Yaskawa INFORM job: A_ROOF_UPPER_0614_2_PAINT_67.JBI

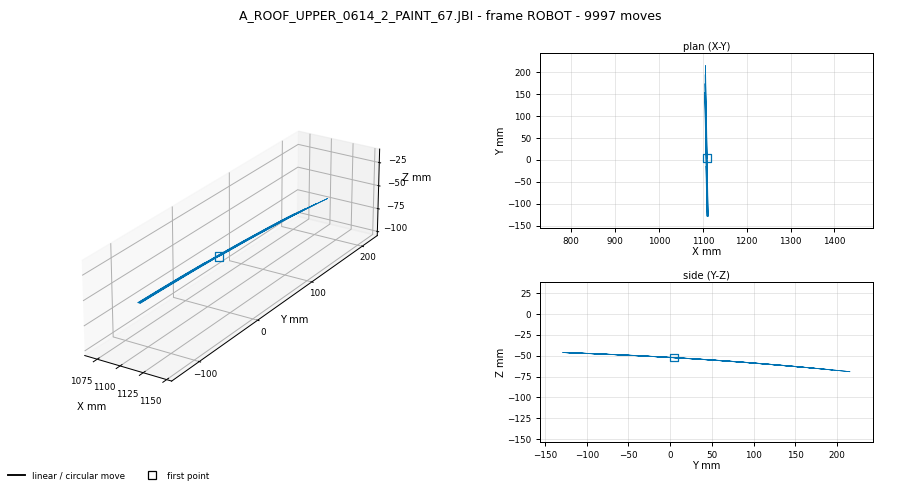
[picture p0: tool path of A_ROOF_UPPER_0614_2_PAINT_67.JBI in frame ROBOT, 9997 of 9997 moves have a stored position in this frame; points joined in program order, loops and branches not executed]
/JOB
//NAME A_ROOF_UPPER_0614_2_PAINT67
//POS
///NPOS 9997,0,0,0,0,0
///TOOL 1
///USER 0
///POSTYPE ROBOT
///RECTAN
///RCONF 1,0,0,0,0,0,0,0,0,0,0,0,0,0,0,0,0,0,0,0,0,0,0,0
C00000=1109.941,4.265,-52.087,179.831,6.526,149.242
C00001=1109.936,4.515,-52.102,179.832,6.531,149.243
C00002=1109.930,4.764,-52.116,179.832,6.536,149.244
C00003=1109.925,5.013,-52.130,179.833,6.541,149.244
C00004=1109.920,5.262,-52.145,179.834,6.545,149.245
C00005=1109.916,5.512,-52.159,179.834,6.550,149.246
C00006=1109.911,5.762,-52.173,179.835,6.554,149.247
C00007=1109.905,6.011,-52.189,179.835,6.559,149.248
C00008=1109.900,6.261,-52.203,179.836,6.564,149.249
C00009=1109.895,6.511,-52.218,179.837,6.568,149.249
C00010=1109.890,6.760,-52.232,179.837,6.573,149.250
C00011=1109.886,7.009,-52.247,179.837,6.577,149.251
C00012=1109.881,7.259,-52.261,179.838,6.581,149.252
C00013=1109.875,7.509,-52.276,179.838,6.586,149.253
C00014=1109.870,7.758,-52.291,179.840,6.590,149.254
C00015=1109.865,8.008,-52.305,179.840,6.595,149.254
C00016=1109.860,8.256,-52.320,179.841,6.600,149.255
C00017=1109.854,8.506,-52.335,179.841,6.605,149.256
C00018=1109.851,8.721,-52.347,179.842,6.609,149.257
C00019=1109.847,8.936,-52.360,179.842,6.613,149.258
C00020=1109.842,9.149,-52.373,179.843,6.616,149.258
C00021=1109.838,9.364,-52.385,179.843,6.620,149.259
C00022=1109.834,9.578,-52.397,179.843,6.625,149.260
C00023=1109.829,9.792,-52.411,179.844,6.628,149.261
C00024=1109.825,10.006,-52.423,179.844,6.632,149.261
C00025=1109.821,10.221,-52.436,179.845,6.636,149.262
C00026=1109.816,10.470,-52.451,179.845,6.640,149.263
C00027=1109.811,10.720,-52.465,179.846,6.645,149.264
C00028=1109.806,10.969,-52.480,179.846,6.649,149.265
C00029=1109.800,11.219,-52.495,179.847,6.654,149.266
C00030=1109.795,11.469,-52.510,179.847,6.659,149.266
C00031=1109.791,11.718,-52.525,179.847,6.663,149.267
C00032=1109.785,11.968,-52.539,179.848,6.667,149.268
C00033=1109.780,12.217,-52.554,179.849,6.672,149.269
C00034=1109.776,12.466,-52.569,179.850,6.676,149.270
C00035=1109.770,12.716,-52.584,179.850,6.681,149.271
C00036=1109.765,12.965,-52.599,179.850,6.685,149.272
C00037=1109.760,13.215,-52.614,179.851,6.689,149.272
C00038=1109.755,13.464,-52.629,179.852,6.694,149.273
C00039=1109.750,13.714,-52.643,179.852,6.699,149.274
C00040=1109.745,13.963,-52.658,179.853,6.703,149.275
C00041=1109.740,14.213,-52.673,179.853,6.707,149.275
C00042=1109.735,14.462,-52.688,179.854,6.712,149.276
C00043=1109.730,14.711,-52.703,179.854,6.716,149.277
C00044=1109.725,14.961,-52.718,179.855,6.721,149.278
C00045=1109.721,15.211,-52.733,179.856,6.725,149.279
C00046=1109.715,15.460,-52.749,179.856,6.729,149.280
C00047=1109.710,15.710,-52.763,179.856,6.734,149.281
C00048=1109.705,15.959,-52.779,179.857,6.738,149.281
C00049=1109.700,16.209,-52.794,179.858,6.743,149.282
C00050=1109.695,16.458,-52.808,179.859,6.747,149.283
C00051=1109.690,16.708,-52.824,179.859,6.751,149.284
C00052=1109.685,16.957,-52.839,179.860,6.756,149.285
C00053=1109.680,17.207,-52.854,179.861,6.760,149.285
C00054=1109.675,17.456,-52.869,179.861,6.765,149.286
C00055=1109.670,17.706,-52.885,179.862,6.770,149.287
C00056=1109.665,17.956,-52.899,179.862,6.773,149.288
C00057=1109.660,18.205,-52.914,179.863,6.778,149.288
C00058=1109.655,18.454,-52.929,179.864,6.782,149.289
C00059=1109.650,18.704,-52.945,179.864,6.787,149.290
C00060=1109.645,18.953,-52.959,179.865,6.790,149.291
C00061=1109.639,19.203,-52.975,179.865,6.795,149.292
C00062=1109.635,19.452,-52.990,179.866,6.799,149.292
C00063=1109.630,19.702,-53.006,179.867,6.804,149.293
C00064=1109.625,19.951,-53.021,179.867,6.809,149.294
C00065=1109.620,20.201,-53.036,179.868,6.812,149.295
C00066=1109.615,20.450,-53.051,179.868,6.817,149.296
C00067=1109.610,20.700,-53.066,179.869,6.821,149.296
C00068=1109.605,20.949,-53.081,179.871,6.826,149.297
C00069=1109.600,21.199,-53.097,179.870,6.830,149.298
C00070=1109.596,21.448,-53.112,179.872,6.834,149.298
C00071=1109.590,21.697,-53.128,179.872,6.839,149.299
C00072=1109.584,21.947,-53.143,179.873,6.843,149.300
C00073=1109.580,22.196,-53.158,179.874,6.848,149.301
C00074=1109.575,22.411,-53.171,179.874,6.851,149.301
C00075=1109.572,22.625,-53.184,179.875,6.855,149.302
C00076=1109.567,22.840,-53.197,179.875,6.858,149.303
C00077=1109.562,23.053,-53.211,179.876,6.863,149.303
C00078=1109.559,23.267,-53.224,179.877,6.866,149.304
C00079=1109.555,23.482,-53.238,179.877,6.869,149.305
C00080=1109.549,23.696,-53.250,179.878,6.873,149.305
C00081=1109.546,23.910,-53.263,179.878,6.876,149.306
C00082=1109.540,24.159,-53.279,179.879,6.881,149.307
C00083=1109.536,24.409,-53.295,179.880,6.885,149.307
C00084=1109.531,24.658,-53.310,179.881,6.890,149.308
C00085=1109.526,24.908,-53.326,179.882,6.894,149.309
C00086=1109.520,25.157,-53.341,179.882,6.898,149.310
C00087=1109.516,25.407,-53.356,179.883,6.902,149.310
C00088=1109.511,25.656,-53.372,179.884,6.907,149.311
C00089=1109.505,25.906,-53.388,179.885,6.911,149.312
C00090=1109.501,26.155,-53.403,179.885,6.915,149.312
C00091=1109.496,26.405,-53.419,179.886,6.919,149.313
C00092=1109.491,26.654,-53.434,179.887,6.924,149.314
C00093=1109.486,26.903,-53.449,179.888,6.928,149.315
C00094=1109.481,27.153,-53.465,179.888,6.932,149.315
C00095=1109.476,27.402,-53.481,179.889,6.936,149.316
C00096=1109.471,27.652,-53.497,179.890,6.941,149.317
C00097=1109.466,27.901,-53.512,179.891,6.945,149.317
C00098=1109.461,28.151,-53.528,179.892,6.949,149.318
C00099=1109.456,28.400,-53.544,179.892,6.953,149.319
C00100=1109.450,28.650,-53.559,179.893,6.957,149.320
C00101=1109.446,28.900,-53.574,179.894,6.962,149.320
C00102=1109.441,29.149,-53.590,179.895,6.966,149.321
C00103=1109.436,29.398,-53.606,179.895,6.970,149.322
C00104=1109.431,29.647,-53.622,179.896,6.974,149.323
C00105=1109.427,29.897,-53.637,179.897,6.979,149.323
C00106=1109.421,30.146,-53.653,179.898,6.983,149.324
C00107=1109.416,30.396,-53.669,179.899,6.986,149.324
C00108=1109.411,30.645,-53.685,179.899,6.991,149.325
C00109=1109.406,30.895,-53.701,179.900,6.995,149.326
C00110=1109.402,31.144,-53.716,179.901,7.000,149.327
C00111=1109.396,31.394,-53.732,179.902,7.003,149.327
C00112=1109.391,31.643,-53.747,179.903,7.007,149.328
C00113=1109.387,31.893,-53.764,179.904,7.012,149.329
C00114=1109.381,32.142,-53.780,179.905,7.016,149.329
C00115=1109.376,32.392,-53.795,179.905,7.020,149.330
C00116=1109.371,32.641,-53.812,179.906,7.024,149.331
C00117=1109.367,32.890,-53.827,179.907,7.029,149.331
C00118=1109.362,33.140,-53.843,179.908,7.033,149.332
C00119=1109.356,33.390,-53.858,179.909,7.037,149.333
C00120=1109.351,33.638,-53.875,179.910,7.041,149.333
C00121=1109.347,33.888,-53.891,179.911,7.045,149.334
C00122=1109.341,34.138,-53.906,179.912,7.049,149.335
C00123=1109.337,34.387,-53.923,179.913,7.054,149.335
C00124=1109.331,34.637,-53.938,179.913,7.057,149.336
C00125=1109.326,34.886,-53.955,179.914,7.061,149.337
C00126=1109.322,35.136,-53.971,179.915,7.066,149.337
C00127=1109.317,35.385,-53.986,179.916,7.070,149.338
C00128=1109.312,35.634,-54.002,179.917,7.074,149.339
C00129=1109.307,35.884,-54.018,179.918,7.078,149.339
C00130=1109.303,36.098,-54.032,179.918,7.081,149.340
C00131=1109.299,36.312,-54.046,179.919,7.086,149.341
C00132=1109.294,36.526,-54.060,179.920,7.089,149.341
C00133=1109.290,36.740,-54.073,179.921,7.092,149.342
C00134=1109.285,36.954,-54.087,179.922,7.096,149.342
C00135=1109.281,37.168,-54.101,179.923,7.100,149.343
C00136=1109.277,37.382,-54.115,179.924,7.103,149.343
C00137=1109.273,37.596,-54.129,179.924,7.106,149.344
C00138=1109.267,37.846,-54.144,179.925,7.111,149.345
C00139=1109.263,38.095,-54.161,179.926,7.115,149.345
C00140=1109.257,38.345,-54.177,179.927,7.119,149.346
C00141=1109.253,38.594,-54.193,179.928,7.123,149.347
C00142=1109.248,38.843,-54.209,179.929,7.127,149.347
C00143=1109.243,39.093,-54.225,179.930,7.132,149.348
C00144=1109.238,39.342,-54.241,179.930,7.135,149.349
C00145=1109.233,39.592,-54.258,179.932,7.139,149.349
C00146=1109.228,39.841,-54.274,179.933,7.143,149.350
C00147=1109.223,40.091,-54.290,179.934,7.148,149.350
C00148=1109.218,40.339,-54.306,179.935,7.151,149.351
C00149=1109.213,40.590,-54.322,179.936,7.155,149.352
C00150=1109.208,40.839,-54.339,179.937,7.160,149.352
C00151=1109.203,41.088,-54.356,179.938,7.164,149.353
C00152=1109.198,41.338,-54.372,179.938,7.168,149.354
C00153=1109.193,41.587,-54.388,179.939,7.172,149.354
C00154=1109.188,41.837,-54.404,179.940,7.176,149.355
C00155=1109.183,42.086,-54.420,179.942,7.180,149.355
C00156=1109.179,42.335,-54.437,179.943,7.184,149.356
C00157=1109.174,42.585,-54.453,179.944,7.188,149.357
C00158=1109.169,42.834,-54.469,179.945,7.192,149.357
C00159=1109.163,43.083,-54.486,179.946,7.196,149.358
C00160=1109.159,43.333,-54.503,179.947,7.201,149.359
C00161=1109.154,43.583,-54.519,179.948,7.204,149.359
C00162=1109.149,43.832,-54.535,179.949,7.208,149.360
C00163=1109.144,44.081,-54.552,179.950,7.213,149.360
C00164=1109.139,44.331,-54.567,179.951,7.217,149.361
C00165=1109.134,44.580,-54.585,179.951,7.220,149.362
C00166=1109.129,44.830,-54.601,179.953,7.224,149.362
C00167=1109.124,45.079,-54.618,179.954,7.229,149.363
C00168=1109.120,45.328,-54.634,179.955,7.233,149.363
C00169=1109.114,45.578,-54.650,179.956,7.237,149.364
C00170=1109.109,45.827,-54.667,179.957,7.241,149.365
C00171=1109.105,46.077,-54.684,179.958,7.245,149.365
C00172=1109.100,46.326,-54.700,179.959,7.249,149.366
C00173=1109.095,46.575,-54.717,179.960,7.253,149.366
C00174=1109.089,46.825,-54.733,179.961,7.257,149.367
C00175=1109.085,47.074,-54.750,179.962,7.261,149.367
C00176=1109.080,47.324,-54.766,179.963,7.265,149.368
C00177=1109.075,47.573,-54.783,179.964,7.269,149.369
C00178=1109.070,47.822,-54.800,179.966,7.273,149.369
C00179=1109.065,48.072,-54.816,179.966,7.277,149.370
C00180=1109.060,48.321,-54.833,179.968,7.281,149.371
C00181=1109.056,48.570,-54.849,179.969,7.285,149.371
C00182=1109.050,48.820,-54.867,179.970,7.289,149.372
C00183=1109.045,49.069,-54.883,179.971,7.293,149.372
C00184=1109.041,49.318,-54.900,179.972,7.297,149.373
C00185=1109.035,49.569,-54.916,179.973,7.301,149.373
C00186=1109.031,49.782,-54.931,179.974,7.304,149.374
C00187=1109.027,49.996,-54.945,179.975,7.308,149.374
C00188=1109.023,50.210,-54.959,179.976,7.311,149.375
C00189=1109.018,50.424,-54.974,179.977,7.315,149.376
C00190=1109.014,50.638,-54.988,179.978,7.318,149.376
C00191=1109.010,50.852,-55.003,179.979,7.322,149.376
C00192=1109.006,51.066,-55.016,179.980,7.325,149.377
C00193=1109.001,51.280,-55.031,179.981,7.329,149.377
C00194=1108.997,51.530,-55.048,179.982,7.333,149.378
C00195=1108.992,51.779,-55.065,179.983,7.337,149.379
C00196=1108.987,52.028,-55.082,179.984,7.340,149.379
C00197=1108.982,52.278,-55.098,179.985,7.344,149.380
C00198=1108.977,52.527,-55.116,179.986,7.349,149.380
C00199=1108.973,52.776,-55.133,179.988,7.352,149.381
C00200=1108.968,53.025,-55.149,179.989,7.357,149.381
C00201=1108.962,53.275,-55.166,179.989,7.360,149.382
C00202=1108.958,53.524,-55.183,179.991,7.364,149.382
C00203=1108.953,53.774,-55.200,179.992,7.368,149.383
C00204=1108.948,54.023,-55.217,179.994,7.372,149.384
C00205=1108.942,54.273,-55.234,179.995,7.377,149.384
C00206=1108.938,54.522,-55.251,179.995,7.380,149.385
C00207=1108.933,54.771,-55.269,179.997,7.384,149.385
C00208=1108.929,55.021,-55.285,179.998,7.388,149.386
C00209=1108.923,55.270,-55.302,179.999,7.392,149.386
C00210=1108.918,55.520,-55.319,-179.999,7.397,149.387
C00211=1108.913,55.769,-55.336,-179.999,7.400,149.387
C00212=1108.909,56.018,-55.354,-179.997,7.404,149.388
C00213=1108.904,56.268,-55.371,-179.996,7.408,149.389
C00214=1108.899,56.517,-55.387,-179.995,7.412,149.389
C00215=1108.893,56.767,-55.404,-179.994,7.416,149.390
C00216=1108.889,57.015,-55.422,-179.993,7.420,149.390
C00217=1108.884,57.265,-55.439,-179.992,7.424,149.391
C00218=1108.880,57.515,-55.456,-179.990,7.428,149.391
C00219=1108.874,57.764,-55.473,-179.989,7.432,149.392
C00220=1108.870,58.013,-55.490,-179.987,7.436,149.392
C00221=1108.864,58.262,-55.507,-179.986,7.440,149.393
C00222=1108.859,58.512,-55.524,-179.985,7.443,149.394
C00223=1108.855,58.761,-55.542,-179.984,7.448,149.394
C00224=1108.850,59.011,-55.559,-179.983,7.452,149.395
C00225=1108.845,59.260,-55.576,-179.982,7.456,149.395
C00226=1108.840,59.509,-55.593,-179.980,7.460,149.396
C00227=1108.834,59.759,-55.611,-179.980,7.463,149.396
C00228=1108.830,60.008,-55.627,-179.978,7.467,149.397
C00229=1108.825,60.257,-55.645,-179.977,7.472,149.397
C00230=1108.821,60.507,-55.662,-179.975,7.475,149.398
C00231=1108.816,60.756,-55.680,-179.974,7.480,149.399
C00232=1108.810,61.006,-55.697,-179.973,7.484,149.399
C00233=1108.806,61.255,-55.714,-179.972,7.487,149.400
C00234=1108.801,61.504,-55.732,-179.971,7.491,149.400
C00235=1108.796,61.754,-55.749,-179.970,7.495,149.401
C00236=1108.791,62.002,-55.766,-179.968,7.499,149.401
C00237=1108.786,62.252,-55.783,-179.966,7.503,149.402
C00238=1108.781,62.501,-55.801,-179.965,7.507,149.402
C00239=1108.776,62.751,-55.818,-179.964,7.511,149.403
C00240=1108.772,63.000,-55.836,-179.963,7.515,149.403
C00241=1108.766,63.250,-55.853,-179.962,7.519,149.404
C00242=1108.763,63.463,-55.868,-179.961,7.522,149.404
C00243=1108.759,63.678,-55.884,-179.959,7.526,149.405
C00244=1108.755,63.891,-55.898,-179.958,7.529,149.405
C00245=1108.750,64.105,-55.913,-179.957,7.532,149.405
C00246=1108.745,64.319,-55.928,-179.956,7.536,149.406
C00247=1108.742,64.533,-55.944,-179.955,7.539,149.407
C00248=1108.737,64.747,-55.959,-179.954,7.543,149.407
C00249=1108.733,64.961,-55.973,-179.953,7.546,149.407
C00250=1108.728,65.210,-55.991,-179.952,7.550,149.408
C00251=1108.723,65.460,-56.009,-179.951,7.554,149.409
C00252=1108.718,65.709,-56.026,-179.949,7.558,149.409
C00253=1108.714,65.958,-56.044,-179.948,7.562,149.409
C00254=1108.709,66.208,-56.061,-179.946,7.566,149.410
C00255=1108.704,66.457,-56.079,-179.945,7.570,149.410
C00256=1108.699,66.706,-56.097,-179.944,7.573,149.411
C00257=1108.695,66.955,-56.114,-179.943,7.577,149.412
C00258=1108.690,67.205,-56.132,-179.941,7.581,149.412
C00259=1108.685,67.454,-56.150,-179.940,7.585,149.413
C00260=1108.680,67.704,-56.167,-179.939,7.589,149.413
C00261=1108.675,67.953,-56.185,-179.937,7.593,149.414
C00262=1108.670,68.202,-56.203,-179.936,7.598,149.414
C00263=1108.665,68.451,-56.221,-179.935,7.601,149.415
C00264=1108.660,68.701,-56.238,-179.933,7.605,149.415
C00265=1108.655,68.950,-56.256,-179.932,7.609,149.416
C00266=1108.650,69.199,-56.274,-179.931,7.613,149.416
C00267=1108.646,69.448,-56.292,-179.929,7.617,149.417
C00268=1108.641,69.699,-56.309,-179.928,7.621,149.417
C00269=1108.636,69.948,-56.327,-179.926,7.625,149.418
C00270=1108.631,70.197,-56.345,-179.925,7.629,149.418
C00271=1108.626,70.446,-56.363,-179.924,7.632,149.419
C00272=1108.621,70.695,-56.381,-179.923,7.636,149.419
C00273=1108.616,70.945,-56.399,-179.921,7.640,149.420
C00274=1108.611,71.194,-56.416,-179.920,7.644,149.420
C00275=1108.607,71.443,-56.434,-179.919,7.648,149.421
C00276=1108.602,71.692,-56.452,-179.917,7.652,149.421
C00277=1108.597,71.942,-56.470,-179.916,7.656,149.422
C00278=1108.592,72.191,-56.488,-179.914,7.660,149.422
C00279=1108.588,72.441,-56.506,-179.913,7.664,149.423
C00280=1108.583,72.690,-56.524,-179.912,7.668,149.423
C00281=1108.578,72.939,-56.542,-179.911,7.672,149.424
C00282=1108.573,73.188,-56.560,-179.909,7.676,149.424
C00283=1108.568,73.437,-56.578,-179.908,7.680,149.425
C00284=1108.563,73.686,-56.596,-179.906,7.684,149.425
C00285=1108.558,73.936,-56.614,-179.905,7.688,149.426
C00286=1108.554,74.186,-56.632,-179.904,7.692,149.426
C00287=1108.549,74.435,-56.649,-179.902,7.696,149.427
C00288=1108.544,74.684,-56.667,-179.901,7.700,149.427
C00289=1108.539,74.933,-56.687,-179.899,7.704,149.428
C00290=1108.534,75.183,-56.705,-179.898,7.707,149.428
C00291=1108.529,75.432,-56.723,-179.897,7.711,149.429
C00292=1108.525,75.682,-56.741,-179.895,7.715,149.429
C00293=1108.520,75.931,-56.759,-179.894,7.719,149.430
C00294=1108.515,76.180,-56.777,-179.893,7.723,149.430
C00295=1108.510,76.429,-56.795,-179.891,7.727,149.431
C00296=1108.505,76.678,-56.813,-179.889,7.731,149.431
C00297=1108.501,76.928,-56.831,-179.888,7.735,149.432
C00298=1108.496,77.142,-56.847,-179.887,7.738,149.432
C00299=1108.492,77.355,-56.863,-179.886,7.741,149.433
C00300=1108.488,77.570,-56.878,-179.885,7.745,149.433
C00301=1108.483,77.783,-56.894,-179.885,7.748,149.434
C00302=1108.479,77.997,-56.910,-179.884,7.751,149.434
C00303=1108.475,78.211,-56.926,-179.883,7.754,149.435
C00304=1108.472,78.425,-56.941,-179.882,7.757,149.435
C00305=1108.467,78.638,-56.956,-179.881,7.760,149.435
C00306=1108.462,78.888,-56.974,-179.881,7.764,149.436
C00307=1108.457,79.138,-56.993,-179.879,7.768,149.437
C00308=1108.453,79.386,-57.012,-179.879,7.771,149.437
C00309=1108.448,79.635,-57.030,-179.877,7.775,149.438
C00310=1108.443,79.885,-57.048,-179.876,7.779,149.438
C00311=1108.438,80.134,-57.066,-179.875,7.783,149.439
C00312=1108.433,80.384,-57.085,-179.874,7.786,149.439
C00313=1108.428,80.633,-57.103,-179.873,7.790,149.440
C00314=1108.423,80.882,-57.121,-179.872,7.794,149.440
C00315=1108.419,81.132,-57.140,-179.871,7.798,149.441
C00316=1108.414,81.380,-57.158,-179.870,7.801,149.442
C00317=1108.409,81.630,-57.177,-179.869,7.805,149.442
C00318=1108.404,81.879,-57.195,-179.868,7.808,149.443
C00319=1108.400,82.129,-57.213,-179.867,7.813,149.443
C00320=1108.395,82.377,-57.232,-179.865,7.816,149.444
C00321=1108.389,82.627,-57.251,-179.865,7.820,149.444
C00322=1108.385,82.877,-57.269,-179.863,7.824,149.445
C00323=1108.380,83.125,-57.288,-179.863,7.827,149.445
C00324=1108.375,83.375,-57.306,-179.861,7.831,149.446
C00325=1108.370,83.625,-57.325,-179.861,7.835,149.446
C00326=1108.366,83.873,-57.343,-179.859,7.839,149.447
C00327=1108.361,84.122,-57.361,-179.858,7.843,149.448
C00328=1108.356,84.372,-57.381,-179.857,7.846,149.448
C00329=1108.351,84.621,-57.399,-179.856,7.850,149.449
C00330=1108.346,84.870,-57.417,-179.855,7.853,149.449
C00331=1108.342,85.120,-57.437,-179.853,7.857,149.450
C00332=1108.337,85.369,-57.455,-179.852,7.862,149.450
C00333=1108.332,85.617,-57.473,-179.851,7.865,149.451
C00334=1108.327,85.868,-57.492,-179.850,7.869,149.451
C00335=1108.322,86.116,-57.511,-179.848,7.873,149.452
C00336=1108.317,86.365,-57.529,-179.848,7.876,149.452
C00337=1108.312,86.616,-57.548,-179.846,7.880,149.453
C00338=1108.308,86.864,-57.566,-179.845,7.884,149.453
C00339=1108.303,87.114,-57.585,-179.844,7.888,149.454
C00340=1108.298,87.363,-57.604,-179.843,7.892,149.454
C00341=1108.293,87.612,-57.622,-179.841,7.895,149.455
C00342=1108.289,87.862,-57.642,-179.841,7.899,149.455
C00343=1108.284,88.110,-57.660,-179.839,7.903,149.456
C00344=1108.278,88.360,-57.679,-179.838,7.907,149.456
C00345=1108.274,88.609,-57.698,-179.837,7.910,149.457
C00346=1108.269,88.858,-57.716,-179.835,7.914,149.457
C00347=1108.265,89.108,-57.736,-179.834,7.918,149.458
C00348=1108.260,89.357,-57.754,-179.833,7.921,149.458
C00349=1108.255,89.606,-57.773,-179.832,7.925,149.459
C00350=1108.250,89.855,-57.792,-179.830,7.929,149.459
C00351=1108.245,90.104,-57.811,-179.829,7.933,149.460
C00352=1108.241,90.354,-57.830,-179.828,7.937,149.460
C00353=1108.235,90.603,-57.848,-179.826,7.941,149.461
C00354=1108.232,90.817,-57.865,-179.825,7.944,149.461
C00355=1108.228,91.031,-57.881,-179.824,7.947,149.462
C00356=1108.223,91.244,-57.897,-179.823,7.951,149.462
C00357=1108.219,91.458,-57.913,-179.822,7.954,149.463
C00358=1108.215,91.671,-57.929,-179.821,7.957,149.463
C00359=1108.211,91.885,-57.946,-179.820,7.960,149.463
C00360=1108.207,92.100,-57.962,-179.819,7.963,149.464
C00361=1108.203,92.313,-57.978,-179.817,7.967,149.464
C00362=1108.198,92.562,-57.998,-179.816,7.970,149.465
C00363=1108.193,92.811,-58.016,-179.815,7.974,149.465
C00364=1108.188,93.061,-58.036,-179.813,7.978,149.466
C00365=1108.184,93.310,-58.054,-179.812,7.982,149.466
C00366=1108.179,93.559,-58.074,-179.811,7.985,149.467
C00367=1108.174,93.808,-58.092,-179.809,7.989,149.467
C00368=1108.169,94.057,-58.112,-179.808,7.993,149.468
C00369=1108.164,94.307,-58.131,-179.806,7.997,149.468
C00370=1108.160,94.556,-58.150,-179.805,8.001,149.468
C00371=1108.154,94.805,-58.169,-179.804,8.004,149.469
C00372=1108.150,95.054,-58.188,-179.802,8.008,149.469
C00373=1108.145,95.303,-58.207,-179.801,8.012,149.470
C00374=1108.140,95.553,-58.227,-179.799,8.016,149.470
C00375=1108.135,95.802,-58.245,-179.798,8.020,149.471
C00376=1108.131,96.052,-58.265,-179.797,8.023,149.471
C00377=1108.125,96.300,-58.284,-179.795,8.027,149.472
C00378=1108.121,96.550,-58.303,-179.794,8.031,149.472
C00379=1108.117,96.799,-58.323,-179.792,8.035,149.473
C00380=1108.112,97.048,-58.341,-179.790,8.039,149.473
C00381=1108.107,97.297,-58.361,-179.789,8.042,149.473
C00382=1108.102,97.546,-58.380,-179.788,8.046,149.474
C00383=1108.097,97.796,-58.400,-179.786,8.049,149.474
C00384=1108.093,98.044,-58.419,-179.785,8.053,149.475
C00385=1108.088,98.294,-58.438,-179.783,8.057,149.475
C00386=1108.083,98.543,-58.458,-179.781,8.061,149.476
C00387=1108.078,98.792,-58.477,-179.780,8.064,149.476
C00388=1108.074,99.042,-58.496,-179.779,8.068,149.476
C00389=1108.068,99.290,-58.516,-179.777,8.072,149.477
C00390=1108.064,99.540,-58.535,-179.776,8.076,149.477
C00391=1108.060,99.789,-58.554,-179.774,8.080,149.478
C00392=1108.054,100.038,-58.574,-179.772,8.084,149.478
C00393=1108.050,100.288,-58.593,-179.770,8.087,149.478
C00394=1108.044,100.537,-58.612,-179.769,8.090,149.479
C00395=1108.040,100.786,-58.632,-179.768,8.094,149.479
C00396=1108.035,101.035,-58.651,-179.766,8.098,149.480
C00397=1108.030,101.284,-58.670,-179.765,8.102,149.480
C00398=1108.025,101.534,-58.690,-179.763,8.106,149.481
C00399=1108.021,101.783,-58.710,-179.761,8.109,149.481
C00400=1108.016,102.032,-58.728,-179.759,8.113,149.481
C00401=1108.012,102.281,-58.749,-179.758,8.117,149.482
C00402=1108.007,102.530,-58.769,-179.756,8.121,149.482
C00403=1108.002,102.779,-58.788,-179.755,8.124,149.483
C00404=1107.997,103.029,-58.807,-179.753,8.128,149.483
C00405=1107.992,103.279,-58.827,-179.751,8.131,149.483
C00406=1107.987,103.527,-58.846,-179.750,8.135,149.484
C00407=1107.983,103.776,-58.866,-179.748,8.139,149.484
C00408=1107.978,104.026,-58.886,-179.746,8.143,149.484
C00409=1107.973,104.275,-58.906,-179.745,8.147,149.485
C00410=1107.969,104.488,-58.923,-179.743,8.149,149.485
C00411=1107.965,104.702,-58.939,-179.742,8.153,149.485
C00412=1107.961,104.916,-58.956,-179.740,8.156,149.486
C00413=1107.957,105.130,-58.973,-179.739,8.159,149.486
C00414=1107.953,105.343,-58.990,-179.737,8.162,149.486
C00415=1107.949,105.556,-59.007,-179.736,8.165,149.487
C00416=1107.944,105.770,-59.024,-179.735,8.168,149.487
C00417=1107.941,105.984,-59.040,-179.733,8.172,149.487
C00418=1107.936,106.233,-59.061,-179.731,8.175,149.487
C00419=1107.931,106.482,-59.080,-179.729,8.179,149.488
C00420=1107.926,106.731,-59.100,-179.727,8.183,149.488
C00421=1107.922,106.980,-59.120,-179.726,8.186,149.489
C00422=1107.917,107.230,-59.140,-179.724,8.190,149.489
C00423=1107.912,107.479,-59.160,-179.722,8.193,149.489
C00424=1107.907,107.728,-59.179,-179.720,8.197,149.489
C00425=1107.902,107.977,-59.199,-179.719,8.201,149.490
C00426=1107.898,108.226,-59.219,-179.716,8.204,149.490
C00427=1107.893,108.476,-59.239,-179.715,8.208,149.490
C00428=1107.888,108.724,-59.259,-179.713,8.211,149.491
C00429=1107.883,108.974,-59.279,-179.711,8.215,149.491
C00430=1107.879,109.223,-59.299,-179.709,8.219,149.491
C00431=1107.874,109.472,-59.319,-179.707,8.222,149.492
C00432=1107.870,109.721,-59.339,-179.705,8.226,149.492
C00433=1107.865,109.971,-59.359,-179.703,8.230,149.492
C00434=1107.860,110.219,-59.379,-179.701,8.233,149.493
C00435=1107.855,110.468,-59.398,-179.700,8.237,149.493
C00436=1107.851,110.717,-59.419,-179.698,8.241,149.493
C00437=1107.845,110.967,-59.439,-179.696,8.244,149.493
C00438=1107.841,111.216,-59.459,-179.694,8.248,149.494
C00439=1107.836,111.466,-59.479,-179.693,8.251,149.494
C00440=1107.831,111.714,-59.499,-179.691,8.254,149.494
C00441=1107.826,111.964,-59.519,-179.689,8.258,149.495
C00442=1107.822,112.213,-59.539,-179.687,8.261,149.495
C00443=1107.818,112.462,-59.559,-179.685,8.264,149.495
C00444=1107.812,112.711,-59.580,-179.684,8.268,149.496
C00445=1107.808,112.960,-59.600,-179.682,8.272,149.496
C00446=1107.803,113.209,-59.620,-179.680,8.274,149.496
C00447=1107.798,113.459,-59.640,-179.679,8.278,149.497
C00448=1107.793,113.707,-59.660,-179.677,8.282,149.497
C00449=1107.789,113.956,-59.680,-179.676,8.285,149.497
C00450=1107.783,114.206,-59.701,-179.674,8.288,149.497
C00451=1107.779,114.455,-59.721,-179.672,8.292,149.498
C00452=1107.775,114.704,-59.741,-179.670,8.296,149.498
C00453=1107.770,114.953,-59.761,-179.668,8.299,149.498
C00454=1107.765,115.202,-59.781,-179.666,8.302,149.499
C00455=1107.760,115.452,-59.802,-179.665,8.306,149.499
C00456=1107.756,115.701,-59.823,-179.663,8.309,149.499
C00457=1107.751,115.950,-59.842,-179.661,8.312,149.499
C00458=1107.747,116.199,-59.863,-179.660,8.316,149.500
C00459=1107.741,116.448,-59.884,-179.658,8.319,149.500
C00460=1107.737,116.697,-59.904,-179.656,8.322,149.500
C00461=1107.732,116.946,-59.924,-179.654,8.326,149.501
C00462=1107.727,117.195,-59.944,-179.653,8.330,149.501
C00463=1107.722,117.444,-59.965,-179.651,8.332,149.501
C00464=1107.718,117.693,-59.985,-179.649,8.336,149.501
C00465=1107.713,117.942,-60.006,-179.647,8.340,149.502
C00466=1107.709,118.156,-60.023,-179.646,8.342,149.502
C00467=1107.705,118.370,-60.040,-179.645,8.345,149.502
C00468=1107.701,118.583,-60.058,-179.643,8.348,149.503
C00469=1107.697,118.797,-60.076,-179.642,8.351,149.503
C00470=1107.693,119.010,-60.094,-179.640,8.353,149.503
C00471=1107.688,119.224,-60.111,-179.638,8.357,149.503
C00472=1107.685,119.437,-60.128,-179.637,8.360,149.503
C00473=1107.681,119.650,-60.146,-179.635,8.362,149.504
C00474=1107.676,119.900,-60.167,-179.634,8.366,149.504
C00475=1107.671,120.149,-60.187,-179.632,8.369,149.504
C00476=1107.667,120.398,-60.207,-179.630,8.372,149.505
C00477=1107.661,120.647,-60.228,-179.629,8.376,149.505
C00478=1107.657,120.896,-60.249,-179.627,8.379,149.505
C00479=1107.652,121.146,-60.270,-179.625,8.382,149.505
C00480=1107.648,121.395,-60.290,-179.623,8.386,149.506
C00481=1107.643,121.644,-60.311,-179.622,8.389,149.506
C00482=1107.638,121.893,-60.332,-179.620,8.392,149.506
C00483=1107.634,122.142,-60.353,-179.618,8.396,149.507
C00484=1107.629,122.391,-60.374,-179.616,8.399,149.507
C00485=1107.625,122.640,-60.394,-179.615,8.403,149.507
C00486=1107.619,122.889,-60.415,-179.613,8.406,149.507
C00487=1107.615,123.138,-60.435,-179.611,8.409,149.508
C00488=1107.610,123.387,-60.456,-179.609,8.412,149.508
C00489=1107.605,123.636,-60.477,-179.608,8.416,149.508
C00490=1107.601,123.885,-60.497,-179.606,8.420,149.509
C00491=1107.596,124.135,-60.518,-179.604,8.422,149.509
C00492=1107.592,124.384,-60.539,-179.602,8.426,149.509
C00493=1107.587,124.633,-60.561,-179.600,8.430,149.509
C00494=1107.583,124.882,-60.581,-179.599,8.432,149.510
C00495=1107.577,125.131,-60.602,-179.597,8.436,149.510
C00496=1107.573,125.380,-60.622,-179.595,8.439,149.510
C00497=1107.568,125.629,-60.643,-179.594,8.443,149.511
C00498=1107.563,125.878,-60.664,-179.592,8.446,149.511
C00499=1107.558,126.127,-60.685,-179.590,8.450,149.511
C00500=1107.555,126.377,-60.706,-179.588,8.452,149.511
C00501=1107.549,126.626,-60.727,-179.586,8.456,149.512
C00502=1107.544,126.875,-60.748,-179.585,8.460,149.512
C00503=1107.540,127.123,-60.769,-179.583,8.462,149.512
C00504=1107.535,127.373,-60.790,-179.581,8.466,149.512
C00505=1107.531,127.622,-60.810,-179.579,8.469,149.513
C00506=1107.526,127.871,-60.832,-179.578,8.472,149.513
C00507=1107.521,128.120,-60.853,-179.576,8.476,149.513
C00508=1107.517,128.369,-60.874,-179.574,8.479,149.514
C00509=1107.511,128.618,-60.895,-179.572,8.482,149.514
C00510=1107.507,128.867,-60.916,-179.571,8.486,149.514
C00511=1107.502,129.116,-60.937,-179.569,8.490,149.514
C00512=1107.498,129.366,-60.958,-179.567,8.492,149.515
C00513=1107.493,129.614,-60.979,-179.565,8.496,149.515
C00514=1107.488,129.864,-61.000,-179.564,8.500,149.515
C00515=1107.483,130.112,-61.022,-179.562,8.503,149.516
C00516=1107.479,130.361,-61.042,-179.560,8.506,149.516
C00517=1107.474,130.611,-61.064,-179.558,8.509,149.516
C00518=1107.470,130.860,-61.085,-179.556,8.513,149.516
C00519=1107.464,131.109,-61.106,-179.555,8.516,149.517
C00520=1107.460,131.357,-61.127,-179.553,8.519,149.517
C00521=1107.456,131.607,-61.149,-179.551,8.523,149.517
C00522=1107.452,131.820,-61.167,-179.550,8.526,149.518
C00523=1107.448,132.034,-61.185,-179.548,8.529,149.518
C00524=1107.443,132.247,-61.204,-179.547,8.531,149.518
C00525=1107.439,132.460,-61.222,-179.546,8.534,149.518
C00526=1107.435,132.673,-61.240,-179.544,8.537,149.519
C00527=1107.432,132.888,-61.258,-179.542,8.540,149.519
C00528=1107.428,133.101,-61.276,-179.541,8.543,149.519
C00529=1107.423,133.315,-61.294,-179.539,8.546,149.519
C00530=1107.419,133.563,-61.316,-179.537,8.549,149.519
C00531=1107.414,133.813,-61.337,-179.536,8.552,149.520
C00532=1107.409,134.062,-61.359,-179.534,8.556,149.520
C00533=1107.404,134.310,-61.380,-179.532,8.559,149.520
C00534=1107.401,134.560,-61.401,-179.530,8.562,149.521
C00535=1107.396,134.808,-61.423,-179.529,8.566,149.521
C00536=1107.391,135.058,-61.444,-179.527,8.569,149.521
C00537=1107.386,135.306,-61.465,-179.525,8.573,149.521
C00538=1107.381,135.556,-61.487,-179.524,8.576,149.522
C00539=1107.376,135.805,-61.508,-179.522,8.580,149.522
C00540=1107.372,136.053,-61.529,-179.520,8.583,149.522
C00541=1107.368,136.303,-61.552,-179.519,8.586,149.523
C00542=1107.363,136.552,-61.572,-179.516,8.590,149.523
C00543=1107.358,136.801,-61.594,-179.514,8.593,149.523
C00544=1107.354,137.050,-61.616,-179.513,8.596,149.524
C00545=1107.348,137.299,-61.637,-179.511,8.600,149.524
C00546=1107.344,137.548,-61.659,-179.509,8.603,149.524
C00547=1107.340,137.797,-61.680,-179.507,8.607,149.524
C00548=1107.335,138.045,-61.702,-179.506,8.610,149.525
C00549=1107.331,138.295,-61.723,-179.504,8.613,149.525
C00550=1107.326,138.544,-61.745,-179.502,8.617,149.525
C00551=1107.321,138.793,-61.767,-179.501,8.620,149.526
C00552=1107.317,139.042,-61.789,-179.499,8.623,149.526
C00553=1107.311,139.291,-61.810,-179.497,8.627,149.526
C00554=1107.307,139.541,-61.832,-179.495,8.631,149.527
C00555=1107.302,139.789,-61.853,-179.494,8.633,149.527
C00556=1107.297,140.038,-61.875,-179.492,8.637,149.527
C00557=1107.293,140.287,-61.897,-179.490,8.641,149.528
C00558=1107.288,140.536,-61.919,-179.488,8.644,149.528
C00559=1107.284,140.786,-61.940,-179.487,8.647,149.528
C00560=1107.279,141.034,-61.962,-179.485,8.651,149.529
C00561=1107.274,141.283,-61.984,-179.483,8.654,149.529
C00562=1107.270,141.532,-62.006,-179.482,8.657,149.529
C00563=1107.265,141.781,-62.027,-179.480,8.661,149.529
C00564=1107.261,142.030,-62.049,-179.478,8.665,149.530
C00565=1107.256,142.279,-62.071,-179.476,8.668,149.530
C00566=1107.251,142.528,-62.093,-179.475,8.671,149.530
C00567=1107.247,142.777,-62.115,-179.473,8.675,149.531
C00568=1107.242,143.026,-62.137,-179.471,8.678,149.531
C00569=1107.237,143.275,-62.158,-179.469,8.682,149.531
C00570=1107.233,143.524,-62.181,-179.468,8.685,149.532
C00571=1107.228,143.773,-62.202,-179.466,8.689,149.532
C00572=1107.224,144.022,-62.224,-179.464,8.692,149.532
C00573=1107.219,144.271,-62.246,-179.462,8.696,149.533
C00574=1107.214,144.520,-62.268,-179.461,8.699,149.533
C00575=1107.210,144.769,-62.290,-179.459,8.702,149.533
C00576=1107.205,145.018,-62.311,-179.457,8.706,149.534
C00577=1107.200,145.267,-62.334,-179.455,8.710,149.534
C00578=1107.196,145.480,-62.352,-179.454,8.712,149.534
C00579=1107.192,145.694,-62.372,-179.452,8.716,149.535
C00580=1107.188,145.907,-62.390,-179.451,8.719,149.535
C00581=1107.184,146.120,-62.409,-179.449,8.722,149.535
C00582=1107.181,146.334,-62.428,-179.447,8.725,149.535
C00583=1107.176,146.547,-62.447,-179.446,8.728,149.536
C00584=1107.173,146.761,-62.466,-179.444,8.731,149.536
C00585=1107.168,146.974,-62.485,-179.442,8.734,149.536
C00586=1107.164,147.223,-62.507,-179.441,8.738,149.536
C00587=1107.159,147.471,-62.529,-179.439,8.741,149.537
C00588=1107.155,147.721,-62.551,-179.437,8.744,149.537
C00589=1107.150,147.970,-62.573,-179.435,8.748,149.537
C00590=1107.145,148.219,-62.595,-179.433,8.751,149.537
C00591=1107.141,148.467,-62.618,-179.431,8.755,149.538
C00592=1107.136,148.716,-62.640,-179.429,8.758,149.538
C00593=1107.132,148.965,-62.662,-179.427,8.762,149.538
C00594=1107.127,149.215,-62.684,-179.425,8.765,149.539
C00595=1107.123,149.463,-62.707,-179.424,8.768,149.539
C00596=1107.118,149.712,-62.729,-179.421,8.772,149.539
C00597=1107.113,149.962,-62.751,-179.419,8.775,149.539
C00598=1107.108,150.210,-62.773,-179.417,8.779,149.540
C00599=1107.104,150.459,-62.796,-179.415,8.782,149.540
C00600=1107.100,150.708,-62.818,-179.413,8.786,149.540
C00601=1107.094,150.957,-62.840,-179.412,8.789,149.540
C00602=1107.090,151.206,-62.863,-179.410,8.792,149.541
C00603=1107.085,151.455,-62.885,-179.408,8.796,149.541
C00604=1107.080,151.704,-62.907,-179.406,8.799,149.541
C00605=1107.076,151.953,-62.930,-179.404,8.803,149.541
C00606=1107.071,152.202,-62.952,-179.401,8.806,149.541
C00607=1107.067,152.451,-62.975,-179.400,8.808,149.542
C00608=1107.062,152.700,-62.997,-179.398,8.812,149.542
C00609=1107.058,152.949,-63.019,-179.396,8.815,149.542
C00610=1107.053,153.198,-63.042,-179.394,8.819,149.542
C00611=1107.049,153.447,-63.064,-179.391,8.822,149.543
C00612=1107.043,153.695,-63.087,-179.390,8.825,149.543
C00613=1107.039,153.945,-63.109,-179.388,8.829,149.543
C00614=1107.035,154.194,-63.132,-179.386,8.832,149.543
C00615=1107.029,154.442,-63.154,-179.384,8.836,149.544
C00616=1107.026,154.691,-63.177,-179.381,8.839,149.544
C00617=1107.020,154.941,-63.200,-179.380,8.841,149.544
C00618=1107.016,155.189,-63.222,-179.378,8.845,149.544
C00619=1107.011,155.439,-63.245,-179.376,8.848,149.544
C00620=1107.007,155.687,-63.267,-179.374,8.852,149.545
C00621=1107.003,155.936,-63.290,-179.372,8.855,149.545
C00622=1106.997,156.185,-63.312,-179.370,8.858,149.545
C00623=1106.993,156.434,-63.335,-179.368,8.861,149.545
C00624=1106.988,156.683,-63.358,-179.365,8.865,149.545
C00625=1106.984,156.931,-63.380,-179.364,8.867,149.546
C00626=1106.979,157.180,-63.404,-179.361,8.870,149.546
C00627=1106.975,157.430,-63.426,-179.359,8.874,149.546
C00628=1106.970,157.679,-63.449,-179.357,8.877,149.546
C00629=1106.965,157.927,-63.471,-179.355,8.880,149.546
C00630=1106.961,158.176,-63.494,-179.353,8.883,149.546
C00631=1106.957,158.425,-63.517,-179.351,8.887,149.547
C00632=1106.952,158.674,-63.540,-179.349,8.890,149.547
C00633=1106.948,158.923,-63.562,-179.347,8.893,149.547
C00634=1106.943,159.136,-63.582,-179.346,8.895,149.547
C00635=1106.940,159.350,-63.601,-179.343,8.898,149.547
C00636=1106.935,159.563,-63.621,-179.342,8.901,149.547
C00637=1106.931,159.776,-63.641,-179.340,8.903,149.547
C00638=1106.927,159.989,-63.660,-179.338,8.906,149.548
C00639=1106.923,160.203,-63.680,-179.337,8.908,149.548
C00640=1106.920,160.416,-63.699,-179.335,8.912,149.548
C00641=1106.916,160.629,-63.719,-179.333,8.915,149.548
C00642=1106.911,160.878,-63.742,-179.331,8.917,149.548
C00643=1106.906,161.127,-63.765,-179.329,8.920,149.548
C00644=1106.902,161.376,-63.788,-179.327,8.924,149.548
C00645=1106.898,161.625,-63.811,-179.324,8.927,149.549
C00646=1106.893,161.873,-63.833,-179.323,8.929,149.549
C00647=1106.888,162.122,-63.856,-179.321,8.933,149.549
C00648=1106.884,162.371,-63.880,-179.318,8.936,149.549
C00649=1106.880,162.620,-63.903,-179.317,8.939,149.549
C00650=1106.875,162.869,-63.926,-179.314,8.942,149.549
C00651=1106.870,163.118,-63.949,-179.312,8.945,149.549
C00652=1106.866,163.367,-63.972,-179.310,8.948,149.550
C00653=1106.861,163.615,-63.995,-179.308,8.951,149.550
C00654=1106.856,163.864,-64.018,-179.306,8.955,149.550
C00655=1106.852,164.113,-64.041,-179.303,8.958,149.550
C00656=1106.848,164.362,-64.065,-179.302,8.960,149.550
C00657=1106.843,164.611,-64.088,-179.299,8.964,149.550
C00658=1106.838,164.860,-64.111,-179.297,8.967,149.551
C00659=1106.834,165.109,-64.134,-179.295,8.969,149.551
C00660=1106.829,165.358,-64.157,-179.293,8.973,149.551
C00661=1106.825,165.607,-64.181,-179.291,8.976,149.551
C00662=1106.820,165.856,-64.204,-179.289,8.978,149.551
C00663=1106.815,166.104,-64.226,-179.287,8.982,149.551
C00664=1106.811,166.353,-64.250,-179.284,8.985,149.551
C00665=1106.806,166.602,-64.273,-179.283,8.988,149.551
C00666=1106.801,166.851,-64.297,-179.280,8.991,149.551
C00667=1106.797,167.100,-64.320,-179.278,8.994,149.552
C00668=1106.793,167.349,-64.343,-179.276,8.997,149.552
C00669=1106.788,167.598,-64.366,-179.274,9.000,149.552
C00670=1106.783,167.847,-64.389,-179.272,9.003,149.552
C00671=1106.779,168.096,-64.413,-179.270,9.005,149.552
C00672=1106.774,168.344,-64.437,-179.268,9.009,149.552
C00673=1106.770,168.593,-64.460,-179.265,9.012,149.552
C00674=1106.765,168.842,-64.484,-179.263,9.014,149.552
C00675=1106.761,169.091,-64.506,-179.261,9.018,149.553
C00676=1106.756,169.340,-64.530,-179.259,9.021,149.553
C00677=1106.751,169.589,-64.553,-179.257,9.024,149.553
C00678=1106.747,169.837,-64.577,-179.255,9.027,149.553
C00679=1106.742,170.087,-64.600,-179.252,9.030,149.553
C00680=1106.738,170.336,-64.624,-179.251,9.033,149.553
C00681=1106.733,170.585,-64.647,-179.248,9.036,149.553
C00682=1106.729,170.833,-64.671,-179.246,9.039,149.553
C00683=1106.724,171.082,-64.695,-179.244,9.042,149.553
C00684=1106.719,171.331,-64.718,-179.242,9.045,149.554
C00685=1106.716,171.579,-64.741,-179.240,9.047,149.554
C00686=1106.711,171.828,-64.765,-179.238,9.050,149.554
C00687=1106.706,172.077,-64.788,-179.235,9.054,149.554
C00688=1106.702,172.326,-64.812,-179.234,9.056,149.554
C00689=1106.697,172.575,-64.836,-179.231,9.059,149.554
C00690=1106.693,172.789,-64.856,-179.229,9.062,149.554
C00691=1106.688,173.001,-64.876,-179.227,9.064,149.554
C00692=1106.685,173.214,-64.897,-179.226,9.067,149.554
C00693=1106.681,173.427,-64.916,-179.224,9.070,149.554
C00694=1106.678,173.640,-64.937,-179.222,9.072,149.554
C00695=1106.673,173.854,-64.957,-179.220,9.075,149.555
C00696=1106.669,174.066,-64.978,-179.218,9.077,149.555
C00697=1106.666,174.279,-64.998,-179.216,9.080,149.555
C00698=1106.661,174.528,-65.021,-179.214,9.083,149.555
C00699=1106.656,174.777,-65.045,-179.212,9.085,149.555
C00700=1106.652,175.026,-65.069,-179.210,9.088,149.555
C00701=1106.648,175.275,-65.093,-179.207,9.092,149.555
C00702=1106.643,175.524,-65.117,-179.206,9.094,149.555
C00703=1106.639,175.773,-65.140,-179.203,9.097,149.555
C00704=1106.634,176.021,-65.164,-179.201,9.101,149.555
C00705=1106.630,176.270,-65.187,-179.199,9.103,149.556
C00706=1106.624,176.519,-65.212,-179.197,9.106,149.556
C00707=1106.620,176.768,-65.235,-179.194,9.109,149.556
C00708=1106.615,177.016,-65.260,-179.193,9.112,149.556
C00709=1106.612,177.266,-65.284,-179.190,9.115,149.556
C00710=1106.607,177.515,-65.307,-179.188,9.118,149.556
C00711=1106.602,177.763,-65.331,-179.186,9.121,149.556
C00712=1106.598,178.012,-65.355,-179.184,9.124,149.556
C00713=1106.593,178.260,-65.379,-179.181,9.127,149.556
C00714=1106.588,178.509,-65.404,-179.180,9.130,149.557
C00715=1106.584,178.759,-65.427,-179.177,9.133,149.557
C00716=1106.580,179.007,-65.451,-179.175,9.136,149.557
C00717=1106.575,179.256,-65.475,-179.173,9.139,149.557
C00718=1106.571,179.505,-65.499,-179.171,9.142,149.557
C00719=1106.566,179.753,-65.523,-179.168,9.145,149.557
C00720=1106.561,180.002,-65.548,-179.166,9.147,149.557
C00721=1106.557,180.252,-65.571,-179.164,9.151,149.557
C00722=1106.553,180.500,-65.595,-179.162,9.154,149.557
C00723=1106.548,180.748,-65.619,-179.160,9.156,149.557
C00724=1106.544,180.998,-65.643,-179.157,9.160,149.558
C00725=1106.539,181.247,-65.668,-179.155,9.163,149.558
C00726=1106.535,181.495,-65.692,-179.153,9.166,149.558
C00727=1106.530,181.744,-65.716,-179.151,9.168,149.558
C00728=1106.526,181.992,-65.740,-179.148,9.172,149.558
C00729=1106.521,182.242,-65.764,-179.146,9.175,149.558
C00730=1106.517,182.491,-65.788,-179.144,9.177,149.558
C00731=1106.512,182.739,-65.812,-179.141,9.180,149.558
C00732=1106.507,182.988,-65.837,-179.139,9.183,149.558
C00733=1106.503,183.237,-65.862,-179.137,9.186,149.558
C00734=1106.499,183.485,-65.886,-179.135,9.189,149.558
C00735=1106.494,183.734,-65.909,-179.132,9.192,149.558
C00736=1106.489,183.983,-65.934,-179.131,9.194,149.558
C00737=1106.485,184.232,-65.958,-179.128,9.198,149.558
C00738=1106.481,184.481,-65.982,-179.126,9.200,149.559
C00739=1106.476,184.729,-66.007,-179.124,9.203,149.559
C00740=1106.471,184.978,-66.031,-179.121,9.206,149.559
C00741=1106.467,185.227,-66.056,-179.119,9.208,149.559
C00742=1106.462,185.476,-66.080,-179.117,9.212,149.559
C00743=1106.458,185.724,-66.104,-179.114,9.215,149.559
C00744=1106.454,185.973,-66.129,-179.112,9.217,149.559
C00745=1106.449,186.222,-66.153,-179.110,9.220,149.559
C00746=1106.445,186.435,-66.174,-179.108,9.222,149.559
C00747=1106.441,186.648,-66.195,-179.106,9.225,149.559
C00748=1106.437,186.861,-66.216,-179.104,9.227,149.559
C00749=1106.434,187.074,-66.236,-179.102,9.229,149.559
C00750=1106.430,187.287,-66.258,-179.100,9.232,149.559
C00751=1106.426,187.500,-66.279,-179.098,9.235,149.559
C00752=1106.422,187.713,-66.300,-179.096,9.237,149.559
C00753=1106.418,187.926,-66.321,-179.094,9.240,149.559
C00754=1106.414,188.175,-66.345,-179.092,9.242,149.559
C00755=1106.409,188.424,-66.370,-179.090,9.245,149.559
C00756=1106.405,188.672,-66.394,-179.087,9.248,149.559
C00757=1106.400,188.921,-66.419,-179.085,9.250,149.559
C00758=1106.396,189.170,-66.444,-179.083,9.254,149.559
C00759=1106.391,189.418,-66.469,-179.081,9.256,149.559
C00760=1106.387,189.667,-66.493,-179.078,9.259,149.559
C00761=1106.382,189.916,-66.518,-179.076,9.262,149.560
C00762=1106.378,190.165,-66.542,-179.074,9.264,149.560
C00763=1106.373,190.414,-66.567,-179.071,9.268,149.560
C00764=1106.369,190.662,-66.592,-179.069,9.271,149.560
C00765=1106.364,190.911,-66.616,-179.067,9.273,149.560
C00766=1106.360,191.160,-66.641,-179.064,9.276,149.560
C00767=1106.355,191.408,-66.666,-179.062,9.278,149.560
C00768=1106.351,191.657,-66.691,-179.060,9.282,149.560
C00769=1106.346,191.906,-66.715,-179.057,9.285,149.560
C00770=1106.341,192.154,-66.740,-179.055,9.287,149.560
C00771=1106.337,192.403,-66.764,-179.053,9.290,149.560
C00772=1106.333,192.652,-66.790,-179.050,9.293,149.560
C00773=1106.328,192.901,-66.815,-179.049,9.296,149.560
C00774=1106.324,193.149,-66.839,-179.046,9.299,149.560
C00775=1106.319,193.398,-66.865,-179.044,9.301,149.560
C00776=1106.315,193.647,-66.889,-179.042,9.304,149.560
C00777=1106.310,193.896,-66.914,-179.039,9.307,149.560
C00778=1106.306,194.144,-66.939,-179.037,9.310,149.560
C00779=1106.302,194.393,-66.964,-179.035,9.313,149.560
C00780=1106.297,194.642,-66.988,-179.032,9.316,149.560
C00781=1106.293,194.891,-67.014,-179.031,9.318,149.561
C00782=1106.288,195.139,-67.038,-179.028,9.322,149.561
C00783=1106.284,195.388,-67.064,-179.026,9.325,149.561
C00784=1106.279,195.637,-67.089,-179.024,9.327,149.561
C00785=1106.275,195.885,-67.114,-179.021,9.330,149.561
C00786=1106.270,196.134,-67.138,-179.019,9.333,149.561
C00787=1106.266,196.383,-67.164,-179.017,9.336,149.561
C00788=1106.261,196.632,-67.189,-179.015,9.339,149.561
C00789=1106.257,196.880,-67.214,-179.012,9.342,149.561
C00790=1106.252,197.129,-67.239,-179.010,9.345,149.561
C00791=1106.248,197.378,-67.264,-179.008,9.348,149.561
C00792=1106.244,197.626,-67.288,-179.005,9.351,149.561
C00793=1106.239,197.875,-67.314,-179.003,9.353,149.561
C00794=1106.234,198.123,-67.339,-179.001,9.356,149.562
C00795=1106.230,198.372,-67.365,-178.998,9.359,149.562
C00796=1106.225,198.621,-67.389,-178.996,9.362,149.562
C00797=1106.221,198.869,-67.414,-178.994,9.365,149.562
C00798=1106.217,199.118,-67.440,-178.991,9.368,149.562
C00799=1106.212,199.367,-67.465,-178.989,9.371,149.562
C00800=1106.208,199.616,-67.491,-178.987,9.373,149.562
C00801=1106.203,199.865,-67.515,-178.984,9.376,149.562
C00802=1106.200,200.078,-67.537,-178.982,9.378,149.562
C00803=1106.196,200.290,-67.559,-178.980,9.381,149.562
C00804=1106.192,200.503,-67.581,-178.978,9.384,149.562
C00805=1106.188,200.716,-67.602,-178.975,9.386,149.562
C00806=1106.184,200.929,-67.623,-178.973,9.388,149.562
C00807=1106.181,201.142,-67.646,-178.971,9.391,149.562
C00808=1106.177,201.355,-67.668,-178.969,9.393,149.562
C00809=1106.173,201.568,-67.689,-178.967,9.396,149.562
C00810=1106.169,201.817,-67.714,-178.964,9.398,149.561
C00811=1106.164,202.065,-67.740,-178.961,9.401,149.562
C00812=1106.159,202.314,-67.766,-178.958,9.404,149.561
C00813=1106.156,202.563,-67.790,-178.956,9.407,149.561
C00814=1106.151,202.811,-67.815,-178.953,9.410,149.561
C00815=1106.147,203.060,-67.841,-178.951,9.412,149.561
C00816=1106.142,203.308,-67.867,-178.948,9.415,149.561
C00817=1106.138,203.557,-67.892,-178.945,9.418,149.561
C00818=1106.133,203.805,-67.918,-178.943,9.421,149.561
C00819=1106.129,204.055,-67.943,-178.940,9.424,149.561
C00820=1106.124,204.303,-67.968,-178.937,9.426,149.561
C00821=1106.120,204.552,-67.994,-178.934,9.429,149.561
C00822=1106.116,204.800,-68.020,-178.931,9.432,149.561
C00823=1106.111,205.049,-68.045,-178.928,9.435,149.561
C00824=1106.107,205.297,-68.071,-178.925,9.438,149.560
C00825=1106.102,205.546,-68.097,-178.923,9.441,149.561
C00826=1106.097,205.794,-68.122,-178.919,9.444,149.560
C00827=1106.093,206.043,-68.148,-178.916,9.447,149.560
C00828=1106.089,206.292,-68.174,-178.913,9.450,149.560
C00829=1106.084,206.541,-68.200,-178.911,9.453,149.560
C00830=1106.079,206.789,-68.225,-178.908,9.456,149.560
C00831=1106.075,207.038,-68.251,-178.905,9.458,149.560
C00832=1106.071,207.287,-68.277,-178.902,9.461,149.560
C00833=1106.067,207.536,-68.303,-178.898,9.465,149.560
C00834=1106.062,207.784,-68.328,-178.895,9.467,149.559
C00835=1106.057,208.032,-68.354,-178.893,9.471,149.560
C00836=1106.053,208.281,-68.380,-178.890,9.473,149.559
C00837=1106.049,208.530,-68.405,-178.886,9.477,149.559
C00838=1106.043,208.778,-68.431,-178.883,9.480,149.559
C00839=1106.040,209.027,-68.458,-178.880,9.482,149.559
C00840=1106.035,209.275,-68.483,-178.877,9.486,149.559
C00841=1106.031,209.524,-68.509,-178.874,9.489,149.559
C00842=1106.027,209.773,-68.535,-178.871,9.492,149.559
C00843=1106.022,210.021,-68.560,-178.868,9.495,149.559
C00844=1106.017,210.270,-68.587,-178.864,9.499,149.559
C00845=1106.013,210.518,-68.613,-178.862,9.502,149.559
C00846=1106.009,210.767,-68.639,-178.858,9.505,149.559
C00847=1106.005,211.016,-68.665,-178.855,9.508,149.558
C00848=1106.000,211.265,-68.691,-178.852,9.512,149.558
C00849=1105.995,211.513,-68.717,-178.849,9.515,149.558
C00850=1105.991,211.761,-68.743,-178.845,9.518,149.558
C00851=1105.987,212.010,-68.769,-178.843,9.521,149.558
C00852=1105.982,212.259,-68.796,-178.839,9.525,149.558
C00853=1105.978,212.508,-68.821,-178.836,9.528,149.558
C00854=1105.974,212.756,-68.847,-178.833,9.531,149.558
C00855=1105.970,213.005,-68.874,-178.830,9.535,149.558
C00856=1105.965,213.254,-68.900,-178.826,9.539,149.558
C00857=1105.961,213.502,-68.926,-178.823,9.542,149.558
C00858=1105.956,213.736,-68.951,-178.821,9.545,149.558
C00859=1105.952,213.971,-68.976,-178.819,9.548,149.558
C00860=1105.948,214.206,-69.001,-178.817,9.550,149.558
C00861=1105.944,214.442,-69.025,-178.814,9.553,149.558
C00862=1105.940,214.677,-69.050,-178.812,9.557,149.558
C00863=1105.935,214.912,-69.076,-178.810,9.559,149.558
C00864=1105.931,215.147,-69.101,-178.807,9.562,149.558
C00865=1105.927,215.382,-69.125,-178.806,9.565,149.559
C00866=1105.690,205.043,-68.101,-178.927,9.436,149.560
C00867=1105.695,204.794,-68.076,-178.929,9.433,149.561
C00868=1105.699,204.545,-68.050,-178.932,9.430,149.561
C00869=1105.704,204.296,-68.025,-178.935,9.428,149.561
C00870=1105.708,204.048,-67.999,-178.938,9.425,149.561
C00871=1105.713,203.799,-67.973,-178.941,9.422,149.561
C00872=1105.717,203.550,-67.948,-178.943,9.419,149.561
C00873=1105.722,203.302,-67.922,-178.946,9.416,149.561
C00874=1105.726,203.053,-67.897,-178.949,9.413,149.561
C00875=1105.731,202.804,-67.871,-178.952,9.410,149.561
C00876=1105.735,202.556,-67.846,-178.955,9.408,149.561
C00877=1105.740,202.307,-67.820,-178.957,9.405,149.561
C00878=1105.744,202.058,-67.795,-178.960,9.403,149.561
C00879=1105.749,201.810,-67.770,-178.962,9.399,149.561
C00880=1105.753,201.561,-67.744,-178.965,9.397,149.561
C00881=1105.757,201.312,-67.718,-178.968,9.394,149.561
C00882=1105.761,201.064,-67.694,-178.971,9.391,149.562
C00883=1105.767,200.765,-67.663,-178.973,9.388,149.561
C00884=1105.772,200.466,-67.633,-178.976,9.384,149.561
C00885=1105.778,200.166,-67.602,-178.979,9.381,149.562
C00886=1105.783,199.868,-67.572,-178.982,9.377,149.561
C00887=1105.788,199.619,-67.547,-178.985,9.374,149.561
C00888=1105.792,199.371,-67.521,-178.987,9.372,149.562
C00889=1105.797,199.122,-67.496,-178.990,9.369,149.562
C00890=1105.800,198.873,-67.471,-178.992,9.366,149.561
C00891=1105.805,198.625,-67.446,-178.994,9.364,149.561
C00892=1105.810,198.375,-67.421,-178.997,9.360,149.561
C00893=1105.815,198.127,-67.395,-178.999,9.357,149.561
C00894=1105.819,197.878,-67.370,-179.001,9.355,149.561
C00895=1105.823,197.630,-67.346,-179.004,9.352,149.561
C00896=1105.827,197.381,-67.320,-179.006,9.349,149.561
C00897=1105.832,197.132,-67.295,-179.008,9.346,149.561
C00898=1105.837,196.884,-67.269,-179.010,9.343,149.561
C00899=1105.841,196.635,-67.245,-179.013,9.340,149.561
C00900=1105.845,196.386,-67.220,-179.014,9.338,149.561
C00901=1105.850,196.137,-67.195,-179.017,9.334,149.561
C00902=1105.854,195.889,-67.170,-179.020,9.331,149.561
C00903=1105.859,195.640,-67.145,-179.021,9.329,149.561
C00904=1105.863,195.392,-67.119,-179.024,9.326,149.560
C00905=1105.868,195.142,-67.094,-179.026,9.322,149.560
C00906=1105.872,194.894,-67.070,-179.028,9.320,149.560
C00907=1105.877,194.645,-67.044,-179.030,9.317,149.560
C00908=1105.882,194.396,-67.020,-179.033,9.314,149.560
C00909=1105.885,194.148,-66.995,-179.035,9.312,149.560
C00910=1105.890,193.899,-66.970,-179.037,9.308,149.560
C00911=1105.895,193.650,-66.945,-179.040,9.305,149.560
C00912=1105.899,193.402,-66.920,-179.041,9.303,149.560
C00913=1105.903,193.152,-66.895,-179.044,9.300,149.560
C00914=1105.908,192.904,-66.871,-179.046,9.296,149.560
C00915=1105.913,192.656,-66.846,-179.048,9.294,149.560
C00916=1105.917,192.407,-66.821,-179.051,9.291,149.560
C00917=1105.922,192.158,-66.797,-179.053,9.288,149.560
C00918=1105.926,191.909,-66.771,-179.055,9.286,149.560
C00919=1105.930,191.661,-66.747,-179.058,9.282,149.559
C00920=1105.935,191.411,-66.722,-179.060,9.280,149.559
C00921=1105.940,191.163,-66.697,-179.062,9.277,149.559
C00922=1105.944,190.915,-66.672,-179.065,9.274,149.559
C00923=1105.948,190.666,-66.647,-179.067,9.272,149.559
C00924=1105.953,190.417,-66.623,-179.069,9.268,149.559
C00925=1105.957,190.168,-66.598,-179.072,9.265,149.559
C00926=1105.962,189.919,-66.574,-179.074,9.263,149.559
C00927=1105.967,189.671,-66.549,-179.076,9.260,149.559
C00928=1105.970,189.422,-66.524,-179.078,9.258,149.559
C00929=1105.976,189.173,-66.500,-179.080,9.254,149.559
C00930=1105.979,188.924,-66.475,-179.083,9.251,149.559
C00931=1105.984,188.676,-66.450,-179.085,9.249,149.559
C00932=1105.989,188.427,-66.426,-179.087,9.246,149.559
C00933=1105.993,188.178,-66.401,-179.090,9.243,149.559
C00934=1105.998,187.929,-66.377,-179.092,9.240,149.559
C00935=1106.002,187.717,-66.355,-179.094,9.238,149.559
C00936=1106.006,187.503,-66.334,-179.096,9.236,149.559
C00937=1106.009,187.290,-66.314,-179.098,9.233,149.559
C00938=1106.014,187.077,-66.293,-179.100,9.230,149.559
C00939=1106.017,186.864,-66.272,-179.102,9.228,149.559
C00940=1106.021,186.652,-66.250,-179.104,9.226,149.559
C00941=1106.024,186.439,-66.230,-179.106,9.223,149.559
C00942=1106.029,186.225,-66.209,-179.108,9.221,149.558
C00943=1106.033,185.977,-66.185,-179.110,9.218,149.558
C00944=1106.038,185.728,-66.160,-179.112,9.216,149.558
C00945=1106.042,185.479,-66.136,-179.115,9.212,149.558
C00946=1106.046,185.231,-66.111,-179.117,9.209,149.558
C00947=1106.051,184.982,-66.087,-179.119,9.207,149.558
C00948=1106.055,184.733,-66.062,-179.121,9.204,149.558
C00949=1106.060,184.484,-66.038,-179.123,9.202,149.558
C00950=1106.065,184.236,-66.014,-179.126,9.198,149.558
C00951=1106.069,183.987,-65.990,-179.128,9.195,149.558
C00952=1106.074,183.737,-65.965,-179.130,9.193,149.558
C00953=1106.078,183.489,-65.941,-179.133,9.190,149.558
C00954=1106.083,183.241,-65.917,-179.135,9.187,149.558
C00955=1106.087,182.991,-65.892,-179.137,9.184,149.558
C00956=1106.092,182.743,-65.868,-179.140,9.181,149.558
C00957=1106.096,182.494,-65.844,-179.142,9.178,149.558
C00958=1106.101,182.245,-65.820,-179.144,9.176,149.558
C00959=1106.105,181.996,-65.795,-179.146,9.172,149.558
C00960=1106.110,181.747,-65.771,-179.149,9.169,149.557
C00961=1106.114,181.499,-65.747,-179.151,9.167,149.557
C00962=1106.119,181.251,-65.723,-179.153,9.164,149.557
C00963=1106.124,181.001,-65.699,-179.156,9.161,149.557
C00964=1106.128,180.752,-65.675,-179.158,9.158,149.557
C00965=1106.132,180.504,-65.651,-179.160,9.155,149.557
C00966=1106.137,180.255,-65.627,-179.162,9.152,149.557
C00967=1106.142,180.006,-65.603,-179.164,9.149,149.557
C00968=1106.146,179.757,-65.578,-179.167,9.146,149.557
C00969=1106.150,179.508,-65.554,-179.169,9.143,149.557
C00970=1106.155,179.259,-65.531,-179.171,9.141,149.557
C00971=1106.159,179.011,-65.507,-179.173,9.137,149.557
C00972=1106.164,178.763,-65.483,-179.175,9.134,149.556
C00973=1106.169,178.513,-65.459,-179.177,9.132,149.556
C00974=1106.173,178.264,-65.434,-179.180,9.128,149.556
C00975=1106.177,178.016,-65.410,-179.182,9.125,149.556
C00976=1106.182,177.767,-65.387,-179.184,9.123,149.556
C00977=1106.186,177.518,-65.363,-179.186,9.120,149.556
C00978=1106.191,177.269,-65.339,-179.188,9.116,149.556
C00979=1106.195,177.021,-65.315,-179.190,9.114,149.556
C00980=1106.200,176.771,-65.290,-179.193,9.111,149.556
C00981=1106.205,176.522,-65.267,-179.195,9.107,149.555
C00982=1106.209,176.274,-65.243,-179.197,9.105,149.555
C00983=1106.214,176.025,-65.220,-179.199,9.102,149.555
C00984=1106.218,175.777,-65.195,-179.202,9.099,149.555
C00985=1106.223,175.528,-65.172,-179.203,9.096,149.555
C00986=1106.227,175.279,-65.148,-179.206,9.093,149.555
C00987=1106.232,175.030,-65.125,-179.208,9.090,149.555
C00988=1106.236,174.781,-65.100,-179.210,9.087,149.555
C00989=1106.240,174.532,-65.077,-179.212,9.084,149.555
C00990=1106.245,174.284,-65.053,-179.215,9.081,149.555
C00991=1106.249,174.070,-65.033,-179.216,9.078,149.554
C00992=1106.253,173.857,-65.012,-179.218,9.076,149.554
C00993=1106.257,173.644,-64.992,-179.220,9.073,149.554
C00994=1106.261,173.431,-64.972,-179.221,9.071,149.554
C00995=1106.264,173.218,-64.951,-179.223,9.068,149.554
C00996=1106.269,173.005,-64.932,-179.225,9.066,149.554
C00997=1106.273,172.792,-64.911,-179.227,9.064,149.554
C00998=1106.277,172.578,-64.891,-179.229,9.060,149.554
C00999=1106.281,172.330,-64.867,-179.231,9.058,149.554
C01000=1106.286,172.081,-64.844,-179.234,9.055,149.554
C01001=1106.290,171.832,-64.820,-179.235,9.052,149.553
C01002=1106.295,171.583,-64.796,-179.238,9.049,149.553
C01003=1106.299,171.334,-64.773,-179.240,9.046,149.553
C01004=1106.304,171.085,-64.749,-179.242,9.043,149.553
C01005=1106.308,170.837,-64.725,-179.244,9.040,149.553
C01006=1106.312,170.588,-64.703,-179.246,9.037,149.553
C01007=1106.317,170.339,-64.679,-179.248,9.034,149.553
C01008=1106.322,170.090,-64.656,-179.251,9.031,149.553
C01009=1106.326,169.842,-64.632,-179.253,9.028,149.552
C01010=1106.331,169.593,-64.609,-179.255,9.025,149.552
C01011=1106.336,169.344,-64.585,-179.257,9.022,149.552
C01012=1106.340,169.095,-64.562,-179.259,9.019,149.552
C01013=1106.345,168.846,-64.538,-179.261,9.016,149.552
C01014=1106.349,168.597,-64.514,-179.263,9.013,149.552
C01015=1106.354,168.348,-64.491,-179.266,9.010,149.552
C01016=1106.358,168.099,-64.468,-179.268,9.007,149.552
C01017=1106.363,167.850,-64.445,-179.270,9.004,149.552
C01018=1106.368,167.601,-64.422,-179.272,9.001,149.552
C01019=1106.372,167.352,-64.398,-179.274,8.998,149.551
C01020=1106.377,167.103,-64.375,-179.276,8.995,149.551
C01021=1106.381,166.855,-64.351,-179.279,8.992,149.551
C01022=1106.385,166.606,-64.328,-179.280,8.989,149.551
C01023=1106.390,166.357,-64.305,-179.283,8.986,149.551
C01024=1106.395,166.109,-64.282,-179.285,8.983,149.551
C01025=1106.400,165.860,-64.258,-179.287,8.980,149.551
C01026=1106.404,165.611,-64.235,-179.289,8.977,149.550
C01027=1106.409,165.362,-64.212,-179.291,8.974,149.550
C01028=1106.413,165.113,-64.189,-179.293,8.971,149.550
C01029=1106.418,164.864,-64.165,-179.295,8.968,149.550
C01030=1106.423,164.615,-64.142,-179.297,8.964,149.550
C01031=1106.427,164.366,-64.119,-179.299,8.962,149.550
C01032=1106.431,164.117,-64.096,-179.301,8.959,149.550
C01033=1106.436,163.868,-64.073,-179.304,8.955,149.550
C01034=1106.441,163.620,-64.050,-179.305,8.953,149.549
C01035=1106.445,163.371,-64.027,-179.308,8.950,149.549
C01036=1106.450,163.122,-64.003,-179.310,8.946,149.549
C01037=1106.454,162.873,-63.981,-179.312,8.944,149.549
C01038=1106.459,162.624,-63.957,-179.314,8.940,149.549
C01039=1106.464,162.375,-63.935,-179.316,8.937,149.549
C01040=1106.468,162.126,-63.912,-179.318,8.934,149.549
C01041=1106.472,161.877,-63.889,-179.320,8.931,149.548
C01042=1106.478,161.629,-63.866,-179.322,8.928,149.548
C01043=1106.482,161.380,-63.843,-179.324,8.926,149.548
C01044=1106.486,161.131,-63.819,-179.326,8.922,149.548
C01045=1106.490,160.882,-63.797,-179.328,8.919,149.548
C01046=1106.495,160.632,-63.774,-179.331,8.915,149.548
C01047=1106.500,160.420,-63.755,-179.332,8.913,149.547
C01048=1106.503,160.206,-63.735,-179.334,8.910,149.547
C01049=1106.508,159.993,-63.715,-179.336,8.908,149.547
C01050=1106.511,159.780,-63.695,-179.338,8.905,149.547
C01051=1106.514,159.567,-63.676,-179.339,8.903,149.547
C01052=1106.519,159.354,-63.656,-179.342,8.900,149.547
C01053=1106.522,159.141,-63.636,-179.343,8.897,149.547
C01054=1106.527,158.928,-63.617,-179.344,8.894,149.546
C01055=1106.532,158.678,-63.594,-179.347,8.891,149.546
C01056=1106.536,158.429,-63.572,-179.348,8.888,149.546
C01057=1106.541,158.180,-63.548,-179.351,8.885,149.546
C01058=1106.545,157.932,-63.527,-179.353,8.882,149.546
C01059=1106.550,157.683,-63.503,-179.355,8.878,149.546
C01060=1106.554,157.434,-63.480,-179.357,8.876,149.545
C01061=1106.559,157.184,-63.458,-179.359,8.872,149.545
C01062=1106.564,156.936,-63.435,-179.361,8.869,149.545
C01063=1106.568,156.687,-63.412,-179.363,8.865,149.545
C01064=1106.573,156.438,-63.390,-179.365,8.863,149.545
C01065=1106.577,156.189,-63.367,-179.367,8.859,149.544
C01066=1106.582,155.940,-63.345,-179.369,8.856,149.544
C01067=1106.587,155.691,-63.322,-179.371,8.853,149.544
C01068=1106.591,155.443,-63.299,-179.373,8.850,149.544
C01069=1106.595,155.193,-63.277,-179.375,8.846,149.544
C01070=1106.600,154.945,-63.254,-179.377,8.843,149.543
C01071=1106.605,154.695,-63.232,-179.380,8.840,149.543
C01072=1106.609,154.446,-63.208,-179.381,8.837,149.543
C01073=1106.614,154.198,-63.187,-179.383,8.834,149.543
C01074=1106.619,153.949,-63.163,-179.385,8.830,149.543
C01075=1106.623,153.699,-63.141,-179.387,8.827,149.542
C01076=1106.628,153.451,-63.119,-179.389,8.824,149.542
C01077=1106.633,153.202,-63.096,-179.391,8.820,149.542
C01078=1106.637,152.953,-63.073,-179.393,8.817,149.542
C01079=1106.642,152.704,-63.051,-179.395,8.814,149.541
C01080=1106.646,152.455,-63.028,-179.397,8.810,149.541
C01081=1106.651,152.206,-63.006,-179.398,8.807,149.541
C01082=1106.656,151.957,-62.984,-179.401,8.804,149.541
C01083=1106.660,151.708,-62.961,-179.403,8.801,149.541
C01084=1106.664,151.459,-62.939,-179.405,8.797,149.541
C01085=1106.670,151.210,-62.917,-179.407,8.793,149.540
C01086=1106.674,150.961,-62.894,-179.408,8.791,149.540
C01087=1106.679,150.713,-62.873,-179.410,8.787,149.540
C01088=1106.684,150.464,-62.849,-179.412,8.784,149.539
C01089=1106.688,150.214,-62.827,-179.415,8.780,149.539
C01090=1106.693,149.966,-62.805,-179.417,8.777,149.539
C01091=1106.697,149.716,-62.783,-179.419,8.773,149.539
C01092=1106.702,149.468,-62.760,-179.420,8.771,149.538
C01093=1106.707,149.219,-62.738,-179.422,8.767,149.538
C01094=1106.711,148.969,-62.716,-179.424,8.764,149.538
C01095=1106.716,148.720,-62.694,-179.426,8.760,149.538
C01096=1106.720,148.472,-62.671,-179.428,8.756,149.537
C01097=1106.725,148.223,-62.650,-179.430,8.753,149.537
C01098=1106.729,147.974,-62.628,-179.432,8.749,149.537
C01099=1106.734,147.725,-62.606,-179.434,8.746,149.537
C01100=1106.739,147.476,-62.582,-179.436,8.743,149.536
C01101=1106.743,147.227,-62.560,-179.437,8.739,149.536
C01102=1106.748,146.978,-62.539,-179.439,8.736,149.536
C01103=1106.753,146.765,-62.520,-179.441,8.733,149.535
C01104=1106.756,146.551,-62.501,-179.443,8.729,149.535
C01105=1106.761,146.338,-62.482,-179.444,8.727,149.535
C01106=1106.764,146.125,-62.463,-179.446,8.724,149.535
C01107=1106.768,145.911,-62.444,-179.447,8.720,149.534
C01108=1106.772,145.699,-62.425,-179.449,8.717,149.534
C01109=1106.776,145.484,-62.406,-179.450,8.715,149.534
C01110=1106.780,145.272,-62.387,-179.452,8.711,149.534
C01111=1106.784,145.023,-62.365,-179.455,8.708,149.533
C01112=1106.789,144.774,-62.344,-179.456,8.705,149.533
C01113=1106.794,144.524,-62.321,-179.458,8.701,149.533
C01114=1106.799,144.276,-62.299,-179.459,8.697,149.532
C01115=1106.803,144.026,-62.277,-179.461,8.694,149.532
C01116=1106.808,143.778,-62.256,-179.462,8.691,149.532
C01117=1106.812,143.528,-62.234,-179.464,8.687,149.531
C01118=1106.817,143.280,-62.212,-179.466,8.683,149.531
C01119=1106.822,143.031,-62.190,-179.468,8.680,149.531
C01120=1106.826,142.782,-62.168,-179.470,8.677,149.530
C01121=1106.831,142.533,-62.146,-179.471,8.673,149.530
C01122=1106.835,142.284,-62.124,-179.473,8.670,149.530
C01123=1106.840,142.035,-62.103,-179.475,8.666,149.529
C01124=1106.844,141.786,-62.081,-179.476,8.663,149.529
C01125=1106.849,141.537,-62.059,-179.478,8.660,149.529
C01126=1106.854,141.288,-62.037,-179.480,8.656,149.528
C01127=1106.859,141.038,-62.016,-179.482,8.652,149.528
C01128=1106.863,140.789,-61.994,-179.483,8.649,149.528
C01129=1106.868,140.540,-61.972,-179.485,8.646,149.527
C01130=1106.873,140.292,-61.951,-179.487,8.642,149.527
C01131=1106.877,140.042,-61.929,-179.489,8.638,149.527
C01132=1106.882,139.794,-61.907,-179.490,8.636,149.527
C01133=1106.886,139.545,-61.885,-179.492,8.632,149.526
C01134=1106.891,139.295,-61.864,-179.494,8.628,149.526
C01135=1106.896,139.047,-61.842,-179.496,8.626,149.526
C01136=1106.900,138.797,-61.820,-179.498,8.622,149.525
C01137=1106.905,138.549,-61.798,-179.499,8.618,149.525
C01138=1106.910,138.299,-61.776,-179.501,8.615,149.525
C01139=1106.915,138.050,-61.755,-179.503,8.612,149.524
C01140=1106.920,137.801,-61.734,-179.504,8.608,149.524
C01141=1106.923,137.552,-61.712,-179.506,8.605,149.524
C01142=1106.928,137.304,-61.691,-179.508,8.602,149.524
C01143=1106.933,137.054,-61.670,-179.510,8.598,149.523
C01144=1106.937,136.805,-61.648,-179.512,8.595,149.523
C01145=1106.942,136.556,-61.626,-179.514,8.591,149.523
C01146=1106.947,136.307,-61.604,-179.515,8.588,149.522
C01147=1106.952,136.058,-61.583,-179.517,8.585,149.522
C01148=1106.957,135.809,-61.561,-179.519,8.581,149.522
C01149=1106.960,135.560,-61.540,-179.520,8.578,149.521
C01150=1106.965,135.311,-61.519,-179.522,8.575,149.521
C01151=1106.970,135.062,-61.497,-179.524,8.571,149.521
C01152=1106.975,134.813,-61.476,-179.526,8.568,149.521
C01153=1106.980,134.564,-61.454,-179.527,8.564,149.520
C01154=1106.984,134.315,-61.433,-179.529,8.561,149.520
C01155=1106.989,134.066,-61.412,-179.531,8.557,149.520
C01156=1106.993,133.817,-61.390,-179.532,8.554,149.519
C01157=1106.998,133.568,-61.369,-179.534,8.551,149.519
C01158=1107.003,133.319,-61.347,-179.536,8.547,149.519
C01159=1107.007,133.106,-61.329,-179.538,8.545,149.519
C01160=1107.011,132.892,-61.311,-179.539,8.542,149.518
C01161=1107.014,132.679,-61.293,-179.541,8.539,149.518
C01162=1107.018,132.466,-61.274,-179.542,8.536,149.518
C01163=1107.023,132.252,-61.256,-179.544,8.533,149.518
C01164=1107.027,132.038,-61.238,-179.545,8.530,149.517
C01165=1107.031,131.825,-61.220,-179.547,8.527,149.517
C01166=1107.035,131.611,-61.202,-179.548,8.524,149.517
C01167=1107.040,131.363,-61.180,-179.550,8.521,149.517
C01168=1107.045,131.113,-61.159,-179.552,8.518,149.516
C01169=1107.049,130.865,-61.138,-179.554,8.515,149.516
C01170=1107.053,130.615,-61.117,-179.555,8.511,149.516
C01171=1107.059,130.366,-61.096,-179.557,8.507,149.515
C01172=1107.063,130.117,-61.075,-179.559,8.505,149.515
C01173=1107.068,129.868,-61.054,-179.561,8.501,149.515
C01174=1107.073,129.620,-61.032,-179.563,8.497,149.515
C01175=1107.077,129.370,-61.011,-179.564,8.495,149.514
C01176=1107.082,129.121,-60.990,-179.566,8.491,149.514
C01177=1107.087,128.872,-60.969,-179.568,8.488,149.514
C01178=1107.091,128.623,-60.948,-179.569,8.485,149.513
C01179=1107.096,128.374,-60.927,-179.571,8.481,149.513
C01180=1107.101,128.124,-60.905,-179.573,8.478,149.513
C01181=1107.105,127.876,-60.885,-179.575,8.475,149.513
C01182=1107.110,127.626,-60.864,-179.576,8.471,149.512
C01183=1107.114,127.378,-60.843,-179.578,8.467,149.512
C01184=1107.119,127.129,-60.822,-179.580,8.465,149.512
C01185=1107.125,126.879,-60.801,-179.582,8.461,149.512
C01186=1107.128,126.630,-60.780,-179.583,8.457,149.511
C01187=1107.133,126.381,-60.758,-179.585,8.455,149.511
C01188=1107.138,126.132,-60.738,-179.587,8.451,149.511
C01189=1107.143,125.883,-60.717,-179.589,8.448,149.510
C01190=1107.147,125.634,-60.697,-179.590,8.445,149.510
C01191=1107.152,125.385,-60.675,-179.592,8.441,149.510
C01192=1107.157,125.136,-60.655,-179.594,8.438,149.510
C01193=1107.161,124.886,-60.633,-179.596,8.434,149.509
C01194=1107.166,124.637,-60.612,-179.597,8.431,149.509
C01195=1107.171,124.388,-60.592,-179.599,8.427,149.509
C01196=1107.176,124.139,-60.571,-179.601,8.424,149.508
C01197=1107.180,123.891,-60.550,-179.603,8.421,149.508
C01198=1107.185,123.642,-60.530,-179.604,8.417,149.508
C01199=1107.190,123.392,-60.509,-179.606,8.414,149.508
C01200=1107.194,123.143,-60.488,-179.608,8.411,149.507
C01201=1107.199,122.894,-60.467,-179.610,8.408,149.507
C01202=1107.203,122.645,-60.446,-179.612,8.404,149.507
C01203=1107.208,122.395,-60.426,-179.613,8.401,149.506
C01204=1107.213,122.146,-60.405,-179.615,8.398,149.506
C01205=1107.218,121.897,-60.384,-179.617,8.394,149.506
C01206=1107.222,121.648,-60.364,-179.618,8.391,149.506
C01207=1107.227,121.399,-60.343,-179.620,8.387,149.505
C01208=1107.232,121.150,-60.322,-179.622,8.384,149.505
C01209=1107.236,120.901,-60.302,-179.624,8.381,149.505
C01210=1107.242,120.652,-60.281,-179.625,8.377,149.504
C01211=1107.246,120.403,-60.261,-179.627,8.374,149.504
C01212=1107.251,120.154,-60.240,-179.629,8.371,149.504
C01213=1107.256,119.905,-60.219,-179.631,8.368,149.504
C01214=1107.260,119.656,-60.199,-179.633,8.364,149.503
C01215=1107.264,119.442,-60.181,-179.634,8.361,149.503
C01216=1107.268,119.229,-60.164,-179.635,8.358,149.503
C01217=1107.272,119.015,-60.145,-179.637,8.356,149.503
C01218=1107.277,118.802,-60.128,-179.638,8.353,149.502
C01219=1107.281,118.588,-60.111,-179.640,8.349,149.502
C01220=1107.284,118.375,-60.093,-179.642,8.347,149.502
C01221=1107.288,118.161,-60.076,-179.643,8.344,149.502
C01222=1107.292,117.948,-60.058,-179.644,8.341,149.501
C01223=1107.297,117.699,-60.038,-179.646,8.337,149.501
C01224=1107.302,117.449,-60.017,-179.648,8.335,149.501
C01225=1107.307,117.200,-59.997,-179.650,8.331,149.501
C01226=1107.311,116.951,-59.976,-179.651,8.327,149.500
C01227=1107.316,116.702,-59.955,-179.653,8.324,149.500
C01228=1107.321,116.453,-59.936,-179.655,8.321,149.500
C01229=1107.325,116.204,-59.915,-179.657,8.317,149.499
C01230=1107.330,115.955,-59.895,-179.659,8.314,149.499
C01231=1107.335,115.705,-59.874,-179.660,8.311,149.499
C01232=1107.340,115.456,-59.854,-179.662,8.307,149.498
C01233=1107.344,115.207,-59.834,-179.664,8.304,149.498
C01234=1107.349,114.958,-59.813,-179.665,8.301,149.498
C01235=1107.354,114.709,-59.793,-179.667,8.297,149.497
C01236=1107.359,114.460,-59.773,-179.669,8.294,149.497
C01237=1107.364,114.211,-59.753,-179.670,8.291,149.497
C01238=1107.368,113.962,-59.732,-179.672,8.287,149.497
C01239=1107.372,113.713,-59.712,-179.674,8.283,149.496
C01240=1107.378,113.463,-59.692,-179.676,8.280,149.496
C01241=1107.382,113.214,-59.671,-179.677,8.277,149.496
C01242=1107.387,112.965,-59.651,-179.679,8.273,149.495
C01243=1107.391,112.716,-59.631,-179.681,8.270,149.495
C01244=1107.396,112.467,-59.611,-179.682,8.267,149.495
C01245=1107.401,112.218,-59.592,-179.684,8.263,149.495
C01246=1107.406,111.969,-59.571,-179.686,8.259,149.494
C01247=1107.411,111.720,-59.550,-179.688,8.256,149.494
C01248=1107.416,111.470,-59.531,-179.689,8.253,149.494
C01249=1107.420,111.221,-59.510,-179.691,8.249,149.493
C01250=1107.425,110.972,-59.491,-179.693,8.246,149.493
C01251=1107.429,110.723,-59.470,-179.695,8.242,149.493
C01252=1107.435,110.474,-59.451,-179.697,8.238,149.492
C01253=1107.439,110.225,-59.431,-179.699,8.235,149.492
C01254=1107.444,109.975,-59.410,-179.701,8.231,149.492
C01255=1107.449,109.726,-59.390,-179.702,8.227,149.491
C01256=1107.453,109.477,-59.370,-179.704,8.224,149.491
C01257=1107.459,109.228,-59.350,-179.706,8.221,149.491
C01258=1107.463,108.979,-59.330,-179.707,8.217,149.491
C01259=1107.468,108.730,-59.310,-179.709,8.214,149.490
C01260=1107.473,108.480,-59.291,-179.711,8.210,149.490
C01261=1107.477,108.231,-59.270,-179.713,8.206,149.490
C01262=1107.482,107.982,-59.251,-179.715,8.203,149.489
C01263=1107.487,107.733,-59.231,-179.717,8.199,149.489
C01264=1107.492,107.484,-59.211,-179.719,8.196,149.489
C01265=1107.496,107.235,-59.191,-179.720,8.192,149.488
C01266=1107.501,106.985,-59.171,-179.722,8.188,149.488
C01267=1107.506,106.736,-59.152,-179.724,8.184,149.488
C01268=1107.511,106.487,-59.131,-179.726,8.181,149.487
C01269=1107.515,106.238,-59.112,-179.728,8.177,149.487
C01270=1107.520,105.988,-59.092,-179.729,8.173,149.487
C01271=1107.524,105.775,-59.076,-179.731,8.170,149.486
C01272=1107.528,105.562,-59.058,-179.732,8.168,149.486
C01273=1107.532,105.348,-59.041,-179.734,8.164,149.486
C01274=1107.536,105.134,-59.024,-179.735,8.161,149.485
C01275=1107.540,104.920,-59.008,-179.737,8.158,149.485
C01276=1107.545,104.707,-58.991,-179.738,8.154,149.485
C01277=1107.548,104.494,-58.974,-179.740,8.152,149.485
C01278=1107.553,104.280,-58.957,-179.741,8.149,149.484
C01279=1107.557,104.030,-58.937,-179.743,8.145,149.484
C01280=1107.563,103.782,-58.918,-179.744,8.141,149.483
C01281=1107.566,103.533,-58.898,-179.746,8.137,149.483
C01282=1107.571,103.283,-58.878,-179.748,8.134,149.483
C01283=1107.576,103.034,-58.859,-179.750,8.130,149.482
C01284=1107.581,102.785,-58.839,-179.751,8.126,149.482
C01285=1107.586,102.535,-58.820,-179.753,8.122,149.482
C01286=1107.591,102.286,-58.800,-179.755,8.119,149.481
C01287=1107.596,102.038,-58.780,-179.756,8.115,149.481
C01288=1107.600,101.788,-58.761,-179.757,8.112,149.480
C01289=1107.605,101.539,-58.741,-179.759,8.108,149.480
C01290=1107.610,101.290,-58.722,-179.761,8.104,149.480
C01291=1107.615,101.040,-58.702,-179.762,8.100,149.479
C01292=1107.619,100.791,-58.683,-179.764,8.096,149.479
C01293=1107.624,100.542,-58.664,-179.766,8.093,149.478
C01294=1107.629,100.293,-58.644,-179.767,8.089,149.478
C01295=1107.634,100.044,-58.625,-179.769,8.086,149.478
C01296=1107.638,99.795,-58.605,-179.770,8.082,149.477
C01297=1107.643,99.545,-58.585,-179.772,8.078,149.477
C01298=1107.648,99.297,-58.566,-179.773,8.074,149.476
C01299=1107.653,99.047,-58.547,-179.775,8.070,149.476
C01300=1107.657,98.797,-58.527,-179.777,8.066,149.475
C01301=1107.662,98.549,-58.508,-179.778,8.063,149.475
C01302=1107.667,98.299,-58.489,-179.779,8.059,149.475
C01303=1107.672,98.051,-58.469,-179.781,8.055,149.474
C01304=1107.677,97.801,-58.450,-179.782,8.051,149.474
C01305=1107.681,97.552,-58.431,-179.784,8.047,149.473
C01306=1107.686,97.303,-58.411,-179.786,8.044,149.473
C01307=1107.691,97.053,-58.392,-179.786,8.040,149.472
C01308=1107.696,96.804,-58.374,-179.788,8.037,149.472
C01309=1107.700,96.554,-58.354,-179.790,8.033,149.471
C01310=1107.706,96.306,-58.335,-179.791,8.029,149.471
C01311=1107.710,96.056,-58.316,-179.793,8.025,149.471
C01312=1107.715,95.807,-58.296,-179.794,8.022,149.470
C01313=1107.720,95.558,-58.277,-179.795,8.018,149.470
C01314=1107.724,95.309,-58.258,-179.797,8.014,149.469
C01315=1107.729,95.060,-58.238,-179.799,8.010,149.469
C01316=1107.734,94.810,-58.220,-179.800,8.006,149.468
C01317=1107.739,94.561,-58.201,-179.801,8.003,149.468
C01318=1107.744,94.311,-58.181,-179.802,7.999,149.467
C01319=1107.748,94.063,-58.162,-179.804,7.995,149.467
C01320=1107.753,93.813,-58.143,-179.806,7.991,149.466
C01321=1107.758,93.564,-58.125,-179.807,7.988,149.466
C01322=1107.763,93.315,-58.105,-179.808,7.984,149.466
C01323=1107.768,93.066,-58.086,-179.810,7.980,149.465
C01324=1107.772,92.816,-58.067,-179.811,7.976,149.465
C01325=1107.777,92.568,-58.047,-179.812,7.972,149.464
C01326=1107.782,92.318,-58.029,-179.813,7.969,149.464
C01327=1107.786,92.105,-58.013,-179.814,7.966,149.463
C01328=1107.790,91.891,-57.996,-179.816,7.962,149.463
C01329=1107.794,91.676,-57.980,-179.817,7.959,149.462
C01330=1107.799,91.463,-57.964,-179.818,7.956,149.462
C01331=1107.802,91.250,-57.947,-179.819,7.953,149.461
C01332=1107.807,91.036,-57.932,-179.820,7.950,149.461
C01333=1107.811,90.822,-57.915,-179.822,7.946,149.461
C01334=1107.815,90.608,-57.899,-179.823,7.943,149.460
C01335=1107.819,90.359,-57.880,-179.824,7.939,149.460
C01336=1107.825,90.110,-57.861,-179.825,7.936,149.459
C01337=1107.829,89.860,-57.842,-179.827,7.932,149.459
C01338=1107.834,89.612,-57.823,-179.828,7.927,149.458
C01339=1107.839,89.362,-57.804,-179.829,7.924,149.458
C01340=1107.844,89.113,-57.785,-179.830,7.920,149.457
C01341=1107.848,88.864,-57.766,-179.831,7.916,149.457
C01342=1107.853,88.614,-57.748,-179.832,7.913,149.456
C01343=1107.858,88.366,-57.729,-179.834,7.909,149.456
C01344=1107.863,88.116,-57.711,-179.835,7.905,149.455
C01345=1107.868,87.867,-57.691,-179.837,7.901,149.455
C01346=1107.872,87.618,-57.672,-179.838,7.898,149.454
C01347=1107.878,87.368,-57.654,-179.839,7.894,149.454
C01348=1107.882,87.119,-57.635,-179.840,7.890,149.453
C01349=1107.887,86.870,-57.617,-179.841,7.886,149.453
C01350=1107.892,86.621,-57.598,-179.843,7.882,149.452
C01351=1107.896,86.371,-57.579,-179.843,7.879,149.452
C01352=1107.901,86.122,-57.560,-179.845,7.875,149.451
C01353=1107.907,85.873,-57.542,-179.846,7.871,149.451
C01354=1107.911,85.624,-57.523,-179.847,7.867,149.450
C01355=1107.916,85.374,-57.504,-179.848,7.864,149.450
C01356=1107.921,85.125,-57.486,-179.850,7.860,149.449
C01357=1107.925,84.876,-57.467,-179.850,7.856,149.448
C01358=1107.931,84.626,-57.449,-179.852,7.852,149.448
C01359=1107.935,84.378,-57.430,-179.853,7.849,149.447
C01360=1107.940,84.128,-57.412,-179.854,7.845,149.447
C01361=1107.944,83.879,-57.393,-179.855,7.841,149.446
C01362=1107.950,83.630,-57.374,-179.856,7.838,149.446
C01363=1107.954,83.380,-57.356,-179.857,7.833,149.445
C01364=1107.959,83.131,-57.337,-179.858,7.830,149.445
C01365=1107.965,82.882,-57.319,-179.859,7.826,149.444
C01366=1107.969,82.632,-57.300,-179.861,7.822,149.444
C01367=1107.973,82.383,-57.282,-179.862,7.818,149.443
C01368=1107.978,82.134,-57.264,-179.863,7.815,149.443
C01369=1107.983,81.884,-57.245,-179.864,7.811,149.442
C01370=1107.988,81.635,-57.226,-179.865,7.807,149.442
C01371=1107.993,81.386,-57.208,-179.866,7.804,149.441
C01372=1107.997,81.136,-57.190,-179.867,7.800,149.440
C01373=1108.003,80.887,-57.171,-179.868,7.796,149.440
C01374=1108.007,80.638,-57.152,-179.869,7.792,149.439
C01375=1108.012,80.389,-57.134,-179.870,7.789,149.439
C01376=1108.017,80.139,-57.116,-179.871,7.785,149.438
C01377=1108.022,79.890,-57.097,-179.873,7.781,149.438
C01378=1108.027,79.641,-57.079,-179.874,7.778,149.437
C01379=1108.032,79.392,-57.061,-179.875,7.773,149.437
C01380=1108.036,79.142,-57.043,-179.876,7.770,149.436
C01381=1108.041,78.893,-57.025,-179.877,7.766,149.435
C01382=1108.046,78.644,-57.006,-179.877,7.762,149.435
C01383=1108.050,78.430,-56.990,-179.878,7.759,149.434
C01384=1108.054,78.216,-56.975,-179.879,7.756,149.434
C01385=1108.059,78.003,-56.959,-179.880,7.753,149.434
C01386=1108.062,77.789,-56.943,-179.881,7.750,149.433
C01387=1108.067,77.575,-56.927,-179.882,7.747,149.432
C01388=1108.071,77.361,-56.912,-179.883,7.743,149.432
C01389=1108.075,77.147,-56.896,-179.884,7.740,149.432
C01390=1108.079,76.933,-56.880,-179.884,7.737,149.431
C01391=1108.084,76.684,-56.862,-179.886,7.733,149.430
C01392=1108.089,76.435,-56.844,-179.887,7.729,149.430
C01393=1108.094,76.186,-56.826,-179.888,7.726,149.430
C01394=1108.099,75.937,-56.808,-179.890,7.722,149.429
C01395=1108.103,75.687,-56.790,-179.891,7.718,149.429
C01396=1108.108,75.437,-56.772,-179.892,7.714,149.428
C01397=1108.113,75.188,-56.754,-179.894,7.710,149.428
C01398=1108.118,74.939,-56.736,-179.896,7.706,149.427
C01399=1108.123,74.690,-56.718,-179.897,7.702,149.427
C01400=1108.127,74.441,-56.699,-179.898,7.698,149.426
C01401=1108.133,74.191,-56.680,-179.900,7.694,149.426
C01402=1108.137,73.942,-56.662,-179.901,7.690,149.425
C01403=1108.142,73.693,-56.644,-179.903,7.686,149.425
C01404=1108.148,73.443,-56.627,-179.904,7.683,149.424
C01405=1108.152,73.194,-56.609,-179.905,7.678,149.424
C01406=1108.157,72.945,-56.591,-179.906,7.674,149.423
C01407=1108.162,72.695,-56.573,-179.908,7.671,149.423
C01408=1108.167,72.446,-56.555,-179.909,7.667,149.422
C01409=1108.172,72.196,-56.537,-179.910,7.662,149.422
C01410=1108.176,71.947,-56.519,-179.912,7.658,149.421
C01411=1108.181,71.698,-56.501,-179.914,7.655,149.421
C01412=1108.186,71.449,-56.483,-179.915,7.650,149.420
C01413=1108.191,71.200,-56.465,-179.916,7.646,149.420
C01414=1108.195,70.951,-56.447,-179.917,7.643,149.419
C01415=1108.200,70.702,-56.429,-179.918,7.639,149.419
C01416=1108.205,70.451,-56.412,-179.920,7.635,149.418
C01417=1108.210,70.202,-56.394,-179.922,7.631,149.418
C01418=1108.215,69.953,-56.376,-179.923,7.627,149.417
C01419=1108.220,69.704,-56.358,-179.924,7.623,149.417
C01420=1108.225,69.455,-56.340,-179.926,7.619,149.416
C01421=1108.229,69.205,-56.322,-179.927,7.615,149.415
C01422=1108.235,68.956,-56.305,-179.928,7.612,149.415
C01423=1108.240,68.706,-56.287,-179.929,7.608,149.415
C01424=1108.244,68.457,-56.269,-179.931,7.603,149.414
C01425=1108.249,68.208,-56.251,-179.932,7.600,149.414
C01426=1108.254,67.959,-56.234,-179.933,7.595,149.413
C01427=1108.259,67.709,-56.216,-179.935,7.591,149.412
C01428=1108.264,67.460,-56.198,-179.936,7.587,149.412
C01429=1108.269,67.210,-56.181,-179.937,7.584,149.411
C01430=1108.274,66.961,-56.163,-179.938,7.580,149.411
C01431=1108.279,66.712,-56.145,-179.940,7.576,149.410
C01432=1108.283,66.463,-56.127,-179.941,7.572,149.410
C01433=1108.288,66.213,-56.110,-179.943,7.568,149.409
C01434=1108.293,65.964,-56.092,-179.944,7.564,149.409
C01435=1108.298,65.715,-56.074,-179.945,7.560,149.408
C01436=1108.303,65.465,-56.057,-179.946,7.557,149.408
C01437=1108.307,65.216,-56.040,-179.947,7.552,149.407
C01438=1108.313,64.967,-56.022,-179.949,7.548,149.407
C01439=1108.316,64.752,-56.006,-179.950,7.545,149.406
C01440=1108.320,64.539,-55.992,-179.951,7.541,149.406
C01441=1108.325,64.325,-55.977,-179.952,7.538,149.406
C01442=1108.329,64.112,-55.962,-179.953,7.535,149.405
C01443=1108.333,63.897,-55.946,-179.954,7.531,149.404
C01444=1108.337,63.683,-55.932,-179.955,7.528,149.404
C01445=1108.342,63.469,-55.917,-179.956,7.525,149.404
C01446=1108.346,63.255,-55.902,-179.957,7.522,149.403
C01447=1108.351,63.006,-55.884,-179.959,7.518,149.403
C01448=1108.355,62.757,-55.866,-179.960,7.513,149.402
C01449=1108.361,62.507,-55.849,-179.961,7.509,149.402
C01450=1108.365,62.259,-55.832,-179.963,7.505,149.401
C01451=1108.370,62.009,-55.814,-179.964,7.501,149.401
C01452=1108.375,61.760,-55.797,-179.965,7.498,149.400
C01453=1108.379,61.510,-55.780,-179.966,7.494,149.399
C01454=1108.385,61.260,-55.763,-179.968,7.490,149.399
C01455=1108.390,61.011,-55.745,-179.969,7.486,149.398
C01456=1108.394,60.762,-55.728,-179.970,7.482,149.398
C01457=1108.400,60.513,-55.710,-179.972,7.477,149.397
C01458=1108.405,60.263,-55.693,-179.972,7.474,149.397
C01459=1108.409,60.015,-55.676,-179.974,7.470,149.396
C01460=1108.414,59.765,-55.658,-179.975,7.466,149.396
C01461=1108.419,59.515,-55.641,-179.976,7.462,149.395
C01462=1108.424,59.266,-55.624,-179.978,7.458,149.395
C01463=1108.429,59.016,-55.606,-179.979,7.454,149.394
C01464=1108.433,58.767,-55.589,-179.980,7.450,149.394
C01465=1108.438,58.518,-55.572,-179.981,7.446,149.393
C01466=1108.444,58.269,-55.555,-179.982,7.442,149.392
C01467=1108.448,58.020,-55.538,-179.984,7.438,149.392
C01468=1108.453,57.770,-55.520,-179.985,7.434,149.391
C01469=1108.458,57.520,-55.504,-179.986,7.431,149.391
C01470=1108.463,57.271,-55.486,-179.987,7.427,149.390
C01471=1108.467,57.022,-55.469,-179.988,7.422,149.390
C01472=1108.473,56.773,-55.452,-179.990,7.418,149.389
C01473=1108.478,56.523,-55.435,-179.991,7.414,149.389
C01474=1108.482,56.274,-55.417,-179.992,7.411,149.388
C01475=1108.488,56.024,-55.400,-179.993,7.407,149.387
C01476=1108.492,55.775,-55.383,-179.994,7.402,149.387
C01477=1108.497,55.525,-55.366,-179.996,7.399,149.386
C01478=1108.502,55.276,-55.350,-179.997,7.394,149.386
C01479=1108.507,55.027,-55.332,-179.998,7.391,149.385
C01480=1108.512,54.777,-55.315,-179.999,7.387,149.385
C01481=1108.517,54.528,-55.298,180.000,7.383,149.384
C01482=1108.522,54.279,-55.282,179.999,7.379,149.384
C01483=1108.527,54.029,-55.264,179.998,7.374,149.383
C01484=1108.532,53.780,-55.248,179.997,7.371,149.382
C01485=1108.536,53.531,-55.230,179.996,7.367,149.382
C01486=1108.541,53.281,-55.213,179.994,7.363,149.381
C01487=1108.546,53.032,-55.197,179.993,7.359,149.381
C01488=1108.552,52.782,-55.180,179.992,7.354,149.380
C01489=1108.556,52.533,-55.163,179.991,7.351,149.380
C01490=1108.561,52.283,-55.146,179.990,7.347,149.379
C01491=1108.566,52.034,-55.129,179.989,7.343,149.378
C01492=1108.571,51.785,-55.113,179.987,7.339,149.378
C01493=1108.576,51.535,-55.095,179.986,7.334,149.377
C01494=1108.581,51.286,-55.079,179.985,7.331,149.377
C01495=1108.585,51.071,-55.064,179.984,7.327,149.376
C01496=1108.589,50.858,-55.049,179.983,7.324,149.376
C01497=1108.593,50.644,-55.035,179.982,7.321,149.375
C01498=1108.597,50.430,-55.021,179.982,7.317,149.375
C01499=1108.602,50.216,-55.006,179.980,7.313,149.374
C01500=1108.606,50.002,-54.992,179.979,7.310,149.374
C01501=1108.610,49.788,-54.977,179.978,7.307,149.373
C01502=1108.614,49.574,-54.964,179.978,7.304,149.373
C01503=1108.620,49.324,-54.946,179.976,7.300,149.372
C01504=1108.625,49.075,-54.930,179.975,7.295,149.372
C01505=1108.629,48.826,-54.913,179.974,7.291,149.371
C01506=1108.634,48.576,-54.897,179.974,7.288,149.370
C01507=1108.640,48.327,-54.880,179.972,7.284,149.370
C01508=1108.644,48.078,-54.863,179.971,7.279,149.369
C01509=1108.649,47.828,-54.846,179.970,7.275,149.369
C01510=1108.654,47.579,-54.830,179.969,7.272,149.368
C01511=1108.659,47.330,-54.813,179.968,7.268,149.367
C01512=1108.663,47.080,-54.796,179.967,7.263,149.367
C01513=1108.668,46.832,-54.780,179.966,7.259,149.366
C01514=1108.674,46.581,-54.763,179.964,7.255,149.366
C01515=1108.678,46.332,-54.747,179.964,7.252,149.365
C01516=1108.683,46.083,-54.730,179.963,7.247,149.364
C01517=1108.688,45.833,-54.714,179.962,7.243,149.364
C01518=1108.694,45.584,-54.697,179.960,7.239,149.363
C01519=1108.698,45.335,-54.680,179.960,7.236,149.363
C01520=1108.703,45.085,-54.664,179.958,7.231,149.362
C01521=1108.708,44.836,-54.648,179.957,7.227,149.361
C01522=1108.713,44.586,-54.631,179.956,7.223,149.361
C01523=1108.718,44.337,-54.614,179.955,7.219,149.360
C01524=1108.723,44.087,-54.598,179.954,7.215,149.360
C01525=1108.728,43.838,-54.582,179.953,7.211,149.359
C01526=1108.733,43.589,-54.565,179.952,7.207,149.358
C01527=1108.737,43.340,-54.549,179.951,7.202,149.358
C01528=1108.743,43.089,-54.532,179.950,7.199,149.357
C01529=1108.748,42.840,-54.516,179.949,7.195,149.357
C01530=1108.752,42.591,-54.499,179.948,7.191,149.356
C01531=1108.757,42.342,-54.483,179.947,7.186,149.355
C01532=1108.762,42.092,-54.467,179.946,7.183,149.355
C01533=1108.767,41.843,-54.451,179.945,7.179,149.354
C01534=1108.772,41.594,-54.434,179.944,7.174,149.353
C01535=1108.777,41.344,-54.418,179.943,7.170,149.353
C01536=1108.782,41.094,-54.401,179.942,7.167,149.352
C01537=1108.787,40.845,-54.384,179.941,7.162,149.352
C01538=1108.792,40.596,-54.369,179.940,7.158,149.351
C01539=1108.797,40.346,-54.352,179.939,7.154,149.350
C01540=1108.802,40.097,-54.337,179.939,7.150,149.350
C01541=1108.807,39.847,-54.320,179.938,7.146,149.349
C01542=1108.812,39.598,-54.304,179.936,7.142,149.348
C01543=1108.816,39.348,-54.288,179.935,7.137,149.348
C01544=1108.822,39.100,-54.271,179.934,7.133,149.347
C01545=1108.826,38.849,-54.255,179.933,7.130,149.347
C01546=1108.831,38.601,-54.239,179.932,7.126,149.346
C01547=1108.836,38.351,-54.223,179.931,7.121,149.345
C01548=1108.841,38.102,-54.207,179.930,7.117,149.345
C01549=1108.846,37.852,-54.191,179.930,7.114,149.344
C01550=1108.851,37.603,-54.175,179.929,7.109,149.343
C01551=1108.855,37.389,-54.161,179.928,7.106,149.343
C01552=1108.860,37.174,-54.147,179.927,7.102,149.342
C01553=1108.864,36.961,-54.133,179.926,7.098,149.342
C01554=1108.868,36.746,-54.119,179.926,7.095,149.341
C01555=1108.873,36.533,-54.106,179.925,7.092,149.340
C01556=1108.877,36.318,-54.092,179.924,7.088,149.340
C01557=1108.881,36.105,-54.078,179.923,7.084,149.339
C01558=1108.885,35.890,-54.064,179.922,7.081,149.339
C01559=1108.891,35.641,-54.048,179.921,7.076,149.338
C01560=1108.895,35.391,-54.032,179.921,7.073,149.337
C01561=1108.901,35.142,-54.016,179.920,7.069,149.337
C01562=1108.906,34.892,-54.000,179.919,7.064,149.336
C01563=1108.911,34.643,-53.984,179.918,7.060,149.335
C01564=1108.915,34.393,-53.968,179.917,7.056,149.335
C01565=1108.920,34.144,-53.951,179.916,7.052,149.334
C01566=1108.926,33.895,-53.936,179.915,7.048,149.333
C01567=1108.930,33.645,-53.921,179.914,7.044,149.333
C01568=1108.935,33.396,-53.904,179.914,7.040,149.332
C01569=1108.940,33.146,-53.888,179.913,7.035,149.331
C01570=1108.945,32.897,-53.873,179.912,7.031,149.331
C01571=1108.950,32.648,-53.856,179.911,7.027,149.330
C01572=1108.955,32.398,-53.840,179.910,7.023,149.329
C01573=1108.960,32.148,-53.825,179.909,7.019,149.329
C01574=1108.965,31.899,-53.808,179.908,7.015,149.328
C01575=1108.970,31.650,-53.793,179.907,7.010,149.327
C01576=1108.975,31.400,-53.778,179.907,7.007,149.327
C01577=1108.980,31.150,-53.762,179.906,7.002,149.326
C01578=1108.985,30.902,-53.745,179.905,6.998,149.325
C01579=1108.990,30.652,-53.730,179.904,6.993,149.324
C01580=1108.995,30.402,-53.714,179.904,6.990,149.324
C01581=1109.000,30.153,-53.699,179.903,6.986,149.323
C01582=1109.005,29.904,-53.683,179.902,6.981,149.323
C01583=1109.009,29.654,-53.667,179.901,6.977,149.322
C01584=1109.015,29.405,-53.651,179.900,6.972,149.321
C01585=1109.020,29.155,-53.635,179.900,6.969,149.320
C01586=1109.024,28.905,-53.620,179.898,6.964,149.320
C01587=1109.030,28.656,-53.604,179.897,6.960,149.319
C01588=1109.035,28.407,-53.588,179.897,6.955,149.318
C01589=1109.040,28.157,-53.572,179.896,6.952,149.317
C01590=1109.044,27.908,-53.557,179.895,6.948,149.317
C01591=1109.050,27.659,-53.542,179.894,6.943,149.316
C01592=1109.054,27.409,-53.526,179.894,6.939,149.315
C01593=1109.060,27.159,-53.510,179.893,6.935,149.315
C01594=1109.064,26.910,-53.495,179.892,6.931,149.314
C01595=1109.069,26.660,-53.479,179.892,6.926,149.313
C01596=1109.075,26.411,-53.464,179.891,6.922,149.312
C01597=1109.080,26.161,-53.448,179.890,6.918,149.312
C01598=1109.084,25.913,-53.432,179.890,6.914,149.311
C01599=1109.089,25.663,-53.416,179.889,6.909,149.310
C01600=1109.094,25.413,-53.401,179.887,6.905,149.310
C01601=1109.099,25.164,-53.386,179.887,6.901,149.309
C01602=1109.105,24.915,-53.370,179.886,6.897,149.308
C01603=1109.109,24.665,-53.354,179.885,6.892,149.307
C01604=1109.114,24.416,-53.339,179.885,6.888,149.306
C01605=1109.119,24.166,-53.324,179.884,6.884,149.306
C01606=1109.125,23.917,-53.308,179.883,6.880,149.305
C01607=1109.129,23.702,-53.296,179.883,6.876,149.305
C01608=1109.133,23.488,-53.282,179.882,6.872,149.304
C01609=1109.137,23.273,-53.268,179.881,6.868,149.303
C01610=1109.141,23.060,-53.255,179.881,6.865,149.303
C01611=1109.146,22.846,-53.242,179.881,6.861,149.302
C01612=1109.150,22.631,-53.229,179.880,6.857,149.301
C01613=1109.154,22.418,-53.216,179.879,6.854,149.301
C01614=1109.159,22.203,-53.202,179.879,6.850,149.300
C01615=1109.163,21.954,-53.187,179.878,6.846,149.299
C01616=1109.169,21.705,-53.172,179.877,6.841,149.298
C01617=1109.174,21.454,-53.156,179.877,6.838,149.298
C01618=1109.178,21.205,-53.141,179.876,6.833,149.297
C01619=1109.184,20.956,-53.126,179.875,6.829,149.296
C01620=1109.188,20.706,-53.111,179.874,6.824,149.295
C01621=1109.194,20.457,-53.095,179.874,6.820,149.295
C01622=1109.198,20.207,-53.080,179.873,6.816,149.294
C01623=1109.203,19.958,-53.064,179.872,6.811,149.293
C01624=1109.209,19.708,-53.049,179.872,6.807,149.292
C01625=1109.214,19.459,-53.034,179.871,6.802,149.292
C01626=1109.219,19.209,-53.019,179.871,6.798,149.291
C01627=1109.224,18.960,-53.004,179.870,6.794,149.290
C01628=1109.228,18.710,-52.988,179.869,6.789,149.289
C01629=1109.233,18.460,-52.974,179.868,6.785,149.288
C01630=1109.239,18.211,-52.958,179.868,6.781,149.288
C01631=1109.243,17.962,-52.943,179.868,6.776,149.287
C01632=1109.249,17.713,-52.928,179.867,6.772,149.286
C01633=1109.254,17.463,-52.913,179.866,6.767,149.285
C01634=1109.259,17.213,-52.898,179.865,6.763,149.285
C01635=1109.264,16.964,-52.883,179.865,6.759,149.284
C01636=1109.269,16.714,-52.867,179.864,6.754,149.283
C01637=1109.274,16.464,-52.852,179.863,6.750,149.282
C01638=1109.278,16.215,-52.837,179.863,6.745,149.281
C01639=1109.284,15.966,-52.822,179.863,6.742,149.280
C01640=1109.289,15.716,-52.808,179.862,6.737,149.280
C01641=1109.294,15.467,-52.792,179.861,6.733,149.279
C01642=1109.299,15.218,-52.777,179.861,6.728,149.278
C01643=1109.304,14.968,-52.762,179.860,6.723,149.277
C01644=1109.309,14.719,-52.747,179.860,6.720,149.276
C01645=1109.314,14.470,-52.732,179.859,6.715,149.275
C01646=1109.319,14.220,-52.717,179.858,6.711,149.275
C01647=1109.323,13.970,-52.702,179.858,6.706,149.274
C01648=1109.329,13.720,-52.687,179.858,6.702,149.273
C01649=1109.334,13.471,-52.672,179.857,6.697,149.272
C01650=1109.338,13.222,-52.657,179.856,6.693,149.271
C01651=1109.344,12.972,-52.642,179.856,6.688,149.271
C01652=1109.349,12.722,-52.627,179.855,6.683,149.270
C01653=1109.354,12.473,-52.613,179.855,6.680,149.269
C01654=1109.359,12.223,-52.597,179.854,6.675,149.268
C01655=1109.364,11.974,-52.583,179.854,6.671,149.267
C01656=1109.369,11.725,-52.568,179.853,6.666,149.266
C01657=1109.374,11.475,-52.553,179.852,6.661,149.266
C01658=1109.379,11.225,-52.538,179.852,6.657,149.265
C01659=1109.384,10.976,-52.524,179.852,6.653,149.264
C01660=1109.389,10.726,-52.508,179.851,6.648,149.263
C01661=1109.394,10.477,-52.494,179.850,6.643,149.262
C01662=1109.399,10.228,-52.479,179.850,6.639,149.261
C01663=1109.403,10.013,-52.466,179.850,6.635,149.260
C01664=1109.408,9.799,-52.453,179.849,6.631,149.260
C01665=1109.412,9.585,-52.441,179.849,6.628,149.259
C01666=1109.417,9.370,-52.428,179.848,6.623,149.258
C01667=1109.421,9.156,-52.416,179.848,6.620,149.258
C01668=1109.425,8.942,-52.403,179.848,6.616,149.257
C01669=1109.429,8.728,-52.390,179.847,6.611,149.256
C01670=1109.434,8.514,-52.378,179.847,6.608,149.255
C01671=1109.438,8.264,-52.363,179.846,6.603,149.254
C01672=1109.444,8.014,-52.348,179.846,6.598,149.254
C01673=1109.449,7.765,-52.333,179.845,6.594,149.253
C01674=1109.454,7.516,-52.319,179.844,6.589,149.252
C01675=1109.459,7.266,-52.305,179.843,6.585,149.251
C01676=1109.464,7.017,-52.289,179.843,6.580,149.250
C01677=1109.469,6.767,-52.275,179.842,6.575,149.249
C01678=1109.474,6.517,-52.261,179.842,6.571,149.248
C01679=1109.479,6.268,-52.246,179.841,6.566,149.248
C01680=1109.484,6.018,-52.231,179.840,6.561,149.247
C01681=1109.489,5.769,-52.217,179.840,6.558,149.246
C01682=1109.494,5.519,-52.201,179.840,6.553,149.245
C01683=1109.499,5.270,-52.187,179.839,6.549,149.244
C01684=1109.504,5.020,-52.173,179.838,6.544,149.244
C01685=1109.509,4.771,-52.159,179.838,6.539,149.243
C01686=1109.514,4.522,-52.144,179.837,6.534,149.242
C01687=1109.519,4.272,-52.130,179.836,6.530,149.241
C01688=1109.525,4.022,-52.115,179.836,6.525,149.240
C01689=1109.530,3.772,-52.101,179.835,6.521,149.239
C01690=1109.534,3.523,-52.086,179.835,6.516,149.238
C01691=1109.539,3.273,-52.071,179.834,6.512,149.238
C01692=1109.544,3.024,-52.057,179.833,6.507,149.237
C01693=1109.549,2.774,-52.043,179.833,6.502,149.236
C01694=1109.555,2.525,-52.029,179.832,6.497,149.235
C01695=1109.559,2.276,-52.014,179.831,6.493,149.234
C01696=1109.564,2.026,-52.000,179.830,6.488,149.234
C01697=1109.569,1.777,-51.985,179.831,6.484,149.233
C01698=1109.574,1.527,-51.971,179.830,6.480,149.232
C01699=1109.579,1.277,-51.957,179.829,6.475,149.231
C01700=1109.585,1.027,-51.942,179.828,6.471,149.230
C01701=1109.590,0.778,-51.928,179.828,6.466,149.229
C01702=1109.595,0.528,-51.914,179.827,6.461,149.228
C01703=1109.600,0.279,-51.899,179.826,6.457,149.228
C01704=1109.605,0.030,-51.884,179.826,6.452,149.227
C01705=1109.610,-0.220,-51.870,179.825,6.448,149.226
C01706=1109.615,-0.470,-51.856,179.824,6.443,149.225
C01707=1109.620,-0.719,-51.842,179.824,6.439,149.224
C01708=1109.625,-0.969,-51.828,179.823,6.434,149.224
C01709=1109.630,-1.218,-51.813,179.823,6.430,149.223
C01710=1109.635,-1.468,-51.799,179.822,6.426,149.222
C01711=1109.640,-1.718,-51.785,179.822,6.421,149.221
C01712=1109.646,-1.967,-51.771,179.821,6.416,149.220
C01713=1109.651,-2.216,-51.757,179.820,6.412,149.220
C01714=1109.656,-2.466,-51.742,179.820,6.407,149.219
C01715=1109.661,-2.716,-51.728,179.819,6.402,149.218
C01716=1109.666,-2.965,-51.715,179.818,6.398,149.217
C01717=1109.670,-3.214,-51.700,179.818,6.393,149.216
C01718=1109.675,-3.464,-51.686,179.817,6.389,149.215
C01719=1109.680,-3.678,-51.674,179.817,6.385,149.215
C01720=1109.685,-3.893,-51.661,179.816,6.382,149.214
C01721=1109.689,-4.107,-51.650,179.815,6.377,149.213
C01722=1109.694,-4.321,-51.638,179.816,6.373,149.212
C01723=1109.698,-4.536,-51.625,179.815,6.370,149.212
C01724=1109.702,-4.750,-51.613,179.814,6.365,149.211
C01725=1109.706,-4.965,-51.601,179.814,6.362,149.210
C01726=1109.711,-5.179,-51.590,179.813,6.358,149.210
C01727=1109.716,-5.429,-51.575,179.813,6.354,149.209
C01728=1109.721,-5.678,-51.561,179.812,6.349,149.208
C01729=1109.726,-5.928,-51.547,179.812,6.344,149.207
C01730=1109.730,-6.177,-51.534,179.811,6.340,149.206
C01731=1109.735,-6.427,-51.519,179.810,6.335,149.206
C01732=1109.741,-6.676,-51.505,179.810,6.330,149.205
C01733=1109.746,-6.926,-51.492,179.809,6.327,149.204
C01734=1109.751,-7.176,-51.477,179.809,6.322,149.203
C01735=1109.757,-7.425,-51.464,179.808,6.317,149.202
C01736=1109.761,-7.674,-51.450,179.808,6.313,149.201
C01737=1109.766,-7.924,-51.436,179.807,6.308,149.201
C01738=1109.772,-8.173,-51.422,179.806,6.304,149.200
C01739=1109.777,-8.423,-51.408,179.806,6.299,149.199
C01740=1109.782,-8.673,-51.394,179.805,6.294,149.198
C01741=1109.786,-8.922,-51.381,179.804,6.290,149.197
C01742=1109.792,-9.172,-51.367,179.804,6.286,149.196
C01743=1109.797,-9.422,-51.353,179.804,6.281,149.196
C01744=1109.802,-9.671,-51.339,179.803,6.277,149.195
C01745=1109.806,-9.920,-51.325,179.802,6.272,149.194
C01746=1109.812,-10.170,-51.312,179.802,6.267,149.193
C01747=1109.817,-10.419,-51.298,179.801,6.263,149.192
C01748=1109.822,-10.669,-51.283,179.801,6.258,149.191
C01749=1109.827,-10.919,-51.270,179.800,6.254,149.191
C01750=1109.832,-11.168,-51.256,179.799,6.249,149.190
C01751=1109.837,-11.418,-51.242,179.800,6.245,149.189
C01752=1109.843,-11.667,-51.229,179.799,6.240,149.188
C01753=1109.847,-11.917,-51.215,179.798,6.236,149.187
C01754=1109.852,-12.167,-51.201,179.798,6.231,149.186
C01755=1109.858,-12.416,-51.188,179.797,6.227,149.185
C01756=1109.862,-12.666,-51.174,179.797,6.222,149.185
C01757=1109.868,-12.915,-51.161,179.796,6.217,149.184
C01758=1109.873,-13.165,-51.147,179.795,6.213,149.183
C01759=1109.877,-13.414,-51.133,179.795,6.209,149.182
C01760=1109.883,-13.664,-51.120,179.795,6.204,149.181
C01761=1109.888,-13.914,-51.106,179.794,6.199,149.180
C01762=1109.893,-14.163,-51.093,179.794,6.195,149.179
C01763=1109.898,-14.413,-51.079,179.793,6.190,149.179
C01764=1109.904,-14.663,-51.065,179.792,6.186,149.178
C01765=1109.908,-14.912,-51.052,179.792,6.181,149.177
C01766=1109.914,-15.162,-51.038,179.791,6.176,149.176
C01767=1109.918,-15.411,-51.025,179.791,6.171,149.175
C01768=1109.924,-15.661,-51.011,179.790,6.167,149.174
C01769=1109.929,-15.910,-50.997,179.790,6.163,149.174
C01770=1109.934,-16.160,-50.984,179.789,6.158,149.173
C01771=1109.939,-16.409,-50.971,179.789,6.154,149.172
C01772=1109.944,-16.659,-50.958,179.788,6.149,149.171
C01773=1109.949,-16.908,-50.944,179.788,6.144,149.170
C01774=1109.955,-17.158,-50.930,179.787,6.140,149.169
C01775=1109.958,-17.372,-50.919,179.787,6.136,149.168
C01776=1109.963,-17.587,-50.907,179.786,6.132,149.168
C01777=1109.967,-17.802,-50.896,179.786,6.128,149.167
C01778=1109.972,-18.016,-50.884,179.786,6.124,149.166
C01779=1109.977,-18.230,-50.872,179.785,6.120,149.165
C01780=1109.981,-18.445,-50.862,179.785,6.116,149.165
C01781=1109.985,-18.659,-50.850,179.785,6.112,149.164
C01782=1109.989,-18.874,-50.838,179.784,6.108,149.163
C01783=1109.994,-19.123,-50.825,179.783,6.103,149.162
C01784=1109.999,-19.373,-50.811,179.783,6.099,149.161
C01785=1110.004,-19.622,-50.798,179.782,6.094,149.161
C01786=1110.010,-19.872,-50.785,179.782,6.090,149.160
C01787=1110.014,-20.121,-50.772,179.782,6.085,149.159
C01788=1110.020,-20.371,-50.758,179.781,6.080,149.158
C01789=1110.025,-20.621,-50.745,179.781,6.076,149.157
C01790=1110.030,-20.870,-50.731,179.780,6.071,149.156
C01791=1110.035,-21.120,-50.719,179.780,6.066,149.155
C01792=1110.041,-21.369,-50.705,179.779,6.062,149.154
C01793=1110.045,-21.619,-50.692,179.779,6.057,149.153
C01794=1110.051,-21.868,-50.678,179.778,6.052,149.152
C01795=1110.056,-22.118,-50.666,179.778,6.047,149.152
C01796=1110.061,-22.368,-50.652,179.777,6.043,149.151
C01797=1110.066,-22.617,-50.640,179.777,6.038,149.150
C01798=1110.071,-22.867,-50.626,179.777,6.033,149.149
C01799=1110.076,-23.116,-50.613,179.776,6.028,149.148
C01800=1110.081,-23.367,-50.600,179.776,6.024,149.147
C01801=1110.087,-23.616,-50.587,179.776,6.019,149.146
C01802=1110.092,-23.865,-50.573,179.776,6.015,149.145
C01803=1110.096,-24.115,-50.560,179.775,6.010,149.144
C01804=1110.102,-24.364,-50.547,179.775,6.005,149.143
C01805=1110.107,-24.614,-50.535,179.774,6.000,149.142
C01806=1110.112,-24.864,-50.521,179.774,5.996,149.141
C01807=1110.118,-25.113,-50.508,179.773,5.991,149.140
C01808=1110.122,-25.363,-50.495,179.773,5.986,149.140
C01809=1110.128,-25.612,-50.482,179.772,5.982,149.139
C01810=1110.133,-25.862,-50.469,179.772,5.976,149.138
C01811=1110.137,-26.112,-50.456,179.773,5.972,149.137
C01812=1110.143,-26.361,-50.443,179.773,5.967,149.136
C01813=1110.148,-26.611,-50.430,179.773,5.963,149.135
C01814=1110.153,-26.861,-50.417,179.773,5.958,149.133
C01815=1110.159,-27.110,-50.404,179.773,5.954,149.133
C01816=1110.163,-27.360,-50.391,179.773,5.950,149.132
C01817=1110.168,-27.610,-50.378,179.773,5.945,149.131
C01818=1110.174,-27.859,-50.365,179.773,5.941,149.130
C01819=1110.179,-28.109,-50.352,179.773,5.937,149.129
C01820=1110.184,-28.358,-50.339,179.773,5.933,149.128
C01821=1110.189,-28.607,-50.326,179.773,5.928,149.127
C01822=1110.194,-28.858,-50.313,179.773,5.924,149.126
C01823=1110.199,-29.107,-50.300,179.772,5.919,149.125
C01824=1110.204,-29.356,-50.288,179.773,5.915,149.124
C01825=1110.209,-29.606,-50.275,179.772,5.910,149.123
C01826=1110.215,-29.856,-50.261,179.772,5.906,149.122
C01827=1110.220,-30.105,-50.249,179.772,5.902,149.121
C01828=1110.225,-30.355,-50.236,179.772,5.898,149.120
C01829=1110.229,-30.605,-50.223,179.772,5.893,149.119
C01830=1110.235,-30.854,-50.210,179.772,5.889,149.118
C01831=1110.239,-31.069,-50.199,179.772,5.885,149.118
C01832=1110.244,-31.284,-50.189,179.771,5.881,149.117
C01833=1110.248,-31.498,-50.178,179.771,5.877,149.116
C01834=1110.253,-31.712,-50.167,179.771,5.873,149.115
C01835=1110.257,-31.927,-50.156,179.771,5.869,149.114
C01836=1110.262,-32.141,-50.145,179.770,5.866,149.114
